(* CODESYS project cryo.library
   Placeholder: ESO LDC Cryo Library
   Title: ESO LDC Cryo Library
   Version: 0.0.0.10
   Company: ESO

Project tree, tasks and I/O mapping:
  libraries: ESO LDC Comm Common Library, 0.2.0.2 (ESO); ESO LDC Comm Serial Library, 0.2.0.2 (ESO); ESO LDC Comm Tcp Library, * (ESO); Tc2_SerialCom, * (Beckhoff Automation GmbH); Tc2_Standard, * (Beckhoff Automation GmbH); Tc2_System, * (Beckhoff Automation GmbH); Tc2_Utilities, * (Beckhoff Automation GmbH); Tc3_Module, * (Beckhoff Automation GmbH); VisuDialogs, * (System); VisuSymbols, 3.5.10.0 (System)
  config/
    CPA_Mapping_SPLC016.xml
    IRATEC_Mapping.xml
    MICADO_Mapping_Evacuation_Local.xml
    SIM_Mapping.xml
  00000000-0000-0000-0000-000000000000|config\CPA_Mapping_SPLC016.xml
  00000000-0000-0000-0000-000000000000|config\IRATEC_Mapping.xml
  00000000-0000-0000-0000-000000000000|config\MICADO_Mapping_Evacuation_Local.xml
  00000000-0000-0000-0000-000000000000|config\SIM_Mapping.xml
  DUTs/
    Enumerations/
      Actuators/
        data type E_CRYO_BIN_ACT_CMD
        data type E_CRYO_BIN_ACT_FEEDBACK
        data type E_CRYO_BIN_ACT_FEEDBACK_STATE
        data type E_CRYO_BIN_ACT_STATE
        data type E_CRYO_BIN_CTRL_ACTION
        data type E_CRYO_BIN_CTRL_STATE
        data type E_CRYO_CTRL_CMD
        data type E_CRYO_CTRL_STATE
        data type E_CRYO_GEN_CTRL_EVENT
      Coolers/
        data type E_CRYO_CPA_ALARM
        data type E_CRYO_CPA_CMDS
        data type E_CRYO_CPA_DIAG_IDX
        data type E_CRYO_CRYOTELGT_CMD
        data type E_CRYO_CRYOTELGT_STATE
      Misc/
        data type E_CRYO_ALARM_IDX
        data type E_CRYO_ALARM_LEVEL
        data type E_CRYO_THLD_MODE
        data type E_CRYO_VOTE
      Pumps/
        data type E_CRYO_PUMP_STATE
        data type E_ECODRY_VERSION
      Sensors/
        data type E_CRYO_SBG232_SENSOR_TYPE
        data type E_CRYO_SENSOR_TYPE_PRESS
        data type E_CRYO_SENSOR_TYPE_TEMP
        data type E_CRYO_SIM_SENS_CMD
      Subsystems/
        Evacuation/
          data type E_CRYO_EVAC_PRESSURES_50000
          data type E_CRYO_EVAC_STATE
          data type E_CRYO_EVAC_STATE_50000
          data type E_CRYO_EVAC_SYS_STATE
          data type E_CRYO_EVAC_VALVES_50000
    Structures/
      Actuators/
        data type T_CRYO_BIN_ACT_STATUS
        data type T_CRYO_BIN_CTRL_STATUS
        data type T_CRYO_GEN_CTRL_STATUS_BASE
      Coolers/
        data type T_CRYO_CPA_ACTIVE_LIMITS
        data type T_CRYO_CPA_CFG
        data type T_CRYO_CPA_CTRL
        data type T_CRYO_CPA_DIAG_CFG
        data type T_CRYO_CPA_INFO
        data type T_CRYO_CPA_STAT
        data type T_CRYO_CRYOTELGT_CFG
        data type T_CRYO_CRYOTELGT_CMD
        data type T_CRYO_CRYOTELGT_CTRL
        data type T_CRYO_CRYOTELGT_STAT
      Misc/
        data type T_CRYO_VOTE_LIST
      Pumps/
        data type T_CRYO_PUMP_ATM2303M_CFG
        data type T_CRYO_PUMP_ATM2303M_STAT
        data type T_CRYO_PUMP_BASE_CFG
        data type T_CRYO_PUMP_BASE_CTRL
        data type T_CRYO_PUMP_BASE_STAT
        data type T_CRYO_PUMP_CMD
        data type T_CRYO_PUMP_HIPACE30_CFG
        data type T_CRYO_PUMP_HIPACE30_STAT
        data type T_CRYO_PUMP_MODBUS_CFG
        data type T_CRYO_PUMP_MODBUS_CTRL
        data type T_CRYO_PUMP_MODBUS_STAT
        data type T_CRYO_PUMP_MVP030_CFG
        data type T_CRYO_PUMP_MVP030_STAT
        data type T_CRYO_PUMP_SERIAL_CFG
      Sensors/
        data type T_CRYO_IOLINK_SENSOR_STATUS
        data type T_CRYO_PRESSURE_STATUS
        data type T_CRYO_PRESSURE_VOTE_STATUS
        data type T_CRYO_PT100_OHM2C_REC
        data type T_CRYO_SBG232_STAT
        data type T_CRYO_SENSOR_STATUS
        data type T_CRYO_SENSOR_STATUS_PRESS
        data type T_CRYO_SENSOR_STATUS_TEMP
        data type T_CRYO_TEMPERATURE_STATUS
      Subsystems/
        Evacuation/
          data type T_CRYO_EVAC_CFG
          data type T_CRYO_EVAC_CFG_50000
          data type T_CRYO_EVAC_CTRL
          data type T_CRYO_EVAC_CTRL_50000
          data type T_CRYO_EVAC_STAT
          data type T_CRYO_EVAC_STAT_50000
          data type T_CRYO_EVAC_SYS_INPUT
          data type T_CRYO_EVACUATION_SYSTEM_STATUS
      System/
        data type T_CRYO_CFG
        data type T_CRYO_CTRL
        data type T_CRYO_LOG
        data type T_CRYO_STAT
  GVLs/
  POUs/
    Actuators/
      function block FB_CRYO_ACTUATOR_CMD [ST]: M_SetPermissionOff, M_SetPermissionOn, M_SetPermissions
      function block FB_CRYO_BIN_ACT [ST]: M_GetFeedback, M_SetCtrlOutput, M_SetStatus
      function block FB_CRYO_BIN_CTRL [ST]: M_Reset, M_SetStatus, M_User_SetAction, M_User_TryRecovery
      function block FB_CRYO_CCC_CTRL [ST]: M_User_SetAction
      function block FB_CRYO_CMD_OVERRIDE [ST]: M_SetAllPermitted, M_SetPermissionOff, M_SetPermissionOn, M_SetPermissions
      function block FB_CRYO_GEN_CTRL_BASE [ST]: M_ActionOffExecute, M_ActionOnExecute, M_ActivitySwitchingOff, M_ActivitySwitchingOn, M_CheckForEvents, M_Configure, M_ControlLoop, M_ExecuteActuators, M_IsError, M_ProcessEvents, M_ReadInputs, M_SetStatus
      function block FB_CRYO_HEATER_CTRL [ST]: M_User_SetAction
      function block FB_CRYO_LN2_CTRL [ST]: M_SetStatus, M_User_SetAction
      function block FB_CRYO_VALVE_CTRL [ST]: M_SetStatus, M_User_SetAction
    Comm/
      function block FB_MODBUS_COMM_CPA [ST]
    Coolers/
      function block FB_CRYO_CPA [ST]: ActivityInitializing, ActivityMonitoring, CheckForEvents, M_ByteSwapFLOAT, M_ByteSwapINT, M_CheckDiagnostics, M_CheckErrors, M_CheckService, M_CheckWarnings, M_ExtractReadings, M_GetModelNumber, M_GetOperatingState, M_SetAlarmText, M_UserConfigure
      function block FB_CRYO_CRYOTELGT [ST]: ActivityInitializing, ActivityInitializing_new, ActivityMonitoring, M_AddCtrlCommands, M_ClearCtrlCommands, M_Configure, M_ExecuteComm, M_FindReadCommand, M_GetCouplerState, M_ReadFromReply, M_StateMachine, M_UpdateStatus, ProcessEvents
      function block FB_RS_COMM_CRYOTELGT [ST]: M_ActionInitExecute, M_ComPortControl, M_Reset
      function block FB_SIM_RS_COMM_CRYOTELGT [ST]: M_ActivityDo, M_GetSimReply
    Pumps/
      function block FB_CRYO_PUMP_ATH2303M [ST]: M_Configure, M_GetSpeed, M_IsReady, M_IsRunning, M_ReadFromReply, M_UpdateStatus
      function block FB_CRYO_PUMP_BASE [ST]: ActivityInitializing, ActivityMonitoring, CheckForEvents, M_Configure, M_ExecuteComm, M_GetCouplerState, M_GetSpeed, M_IsReady, M_IsRunning, M_StateMachine, M_UpdateStatus, ProcessEvents
      function block FB_CRYO_PUMP_ECODRY [ST]: M_Configure, M_ExtractReadings_V01, M_ExtractReadings_V21_22, M_IsReady, M_IsRunning, M_ReadFromReply, M_UpdateStatus
      function block FB_CRYO_PUMP_HIPACE30 [ST]: M_Configure, M_GetSpeed, M_IsReady, M_IsRunning, M_ReadFromReply, M_UpdateStatus
      function block FB_CRYO_PUMP_MODBUS [ST]: ActivityInitializing, ActivityMonitoring, M_ByteSwapFLOAT, M_ByteSwapINT, M_ByteSwapUINT, M_ExecuteComm, M_GetCouplerState, M_ReadFromReply, M_SetCommand
      function block FB_CRYO_PUMP_MVP030 [ST]: M_Configure, M_GetSpeed, M_IsReady, M_IsRunning, M_ReadFromReply, M_UpdateStatus
      function block FB_CRYO_PUMP_SERIAL [ST]: ActivityInitializing, ActivityMonitoring, M_ExecuteComm, M_GetCouplerState, M_PVP_Checksum, M_ReadFromReply
    Sensors/
      function block FB_CRYO_PRESSURE [ST]: M_ReadSensors, M_SetStatus
      function block FB_CRYO_PRESSURE_VOTE [ST]: M_CheckWarnings, M_Configure, M_SetConnected, M_SetStatus, M_SetStatus_Average, M_SetStatus_FirstValid, M_SetStatus_Maximum, M_SetStatus_Minimum, M_SetStatus_XooY, M_SetWarning
      function block FB_CRYO_SBG232 [ST]: M_Configure, M_SetError, M_SetReading, M_UpdateStatus
      function block FB_CRYO_SENSOR_BASE [ST]: M_ReadSensor, M_SetStatus
      function block FB_CRYO_SENSOR_PRESSURE [ST]: M_SetStatus, M_SetStatus_CMR_361, M_SetStatus_PKR_250, M_SetStatus_PKR_360, M_SetStatus_WRG_D_NW25
      function block FB_CRYO_SENSOR_TEMPERATURE [ST]: M_GetRamp, M_PT100_Interpolate_Ohm2C, M_PT100_Ohm2C, M_SetStatus, M_SetStatus_PT100
      function block FB_CRYO_TEMPERATURE [ST]: M_GetTemperatureFromLakeshore, M_ReadSensors, M_SetStatus
    Simulation/
      function block FB_CRYO_SIM_CTRL [ST]
      function block FB_CRYO_SIM_PRESSURE [ST]: M_bit2mbar, M_mbar2bit, M_RampTo, M_SetValue, M_StartCurve, M_StartRamp, M_Stop
      function block FB_CRYO_SIM_SBG232 [ST]
      function block FB_CRYO_SIM_SINE [ST]
      function block FB_CRYO_SIM_TEMPERATURE [ST]: M_bit2degK, M_degK2bit, M_RampTo, M_SetValue, M_StartRamp, M_StartSine, M_Stop
      function block FB_SIM_MODBUS_COMM_CPA [ST]: M_GetSimReply
    Subsystems/
      Evacuation/
        function block FB_CRYO_EVAC_BASE [ST]: M_Activity_ClosingValve, M_Activity_DelayBeforeStoppingPumps, M_Activity_Evacuating, M_Activity_Off, M_Activity_OpeningValve, M_Activity_StartingRoughingPump, M_Activity_StartingTurboPump, M_Activity_StoppingRoughingPump, M_Activity_StoppingTurboPump, M_Activity_WaitingCryoVacuum, M_Activity_WaitingPrevacuum, M_Activity_WaitingTurboPump2Stop, M_Configure, M_ExecuteControllers, M_GotoOff, M_ReadSensors, M_SetError, M_SetLabels, M_StateMachine, M_UpdateStatus
        function block FB_CRYO_EVAC_BASE_50000 [ST]: M_ActionExecute, M_Activity_ClosingAllValves, M_Activity_ClosingValve, M_Activity_DelayBeforeStoppingPumps, M_Activity_Evacuating, M_Activity_Off, M_Activity_OpeningValve, M_Activity_StartingPVP, M_Activity_StartingTMP, M_Activity_StoppingPVP, M_Activity_StoppingTMP, M_Activity_Waiting2Pressures, M_Activity_WaitingPressure, M_Activity_WaitingTMP2Stop, M_Configure, M_ExecuteControllers, M_ReadSensors, M_SetError, M_SetLabels, M_SetNextState, M_StateMachine, M_UpdateStatus
        function block FB_CRYO_EVACUATION_SYSTEM [ST]: M_CheckErrors, M_PumpCtrl, M_SetStatus, M_SetValveCommand, M_StateMachine, M_TrgValveClosure, M_User_TryRecovery
      Examples/
        Evacuation/
          function block FB_CRYO_EVAC_ECODRY_ATH2303M [ST]: M_Configure, M_ExecuteControllers
          function block FB_CRYO_EVAC_MICADO [ST]: M_Configure, M_ExecuteControllers
          function block FB_CRYO_EVAC_PDS [ST]: M_Configure, M_ExecuteControllers
          function block FB_SIM_MICADO_PUMPS [ST]
          function block FB_SIM_MICADO_VALVES [ST]
        LN2_Precooling/
          function block FB_CRYO_LN2_PRECOOL [ST]: M_ActionOffExecute, M_ActionOnExecute, M_ActivitySwitchingOff, M_ActivitySwitchingOn, M_Configure, M_ControlLoop, M_ExecuteActuators, M_IsError, M_SetStatus
          function block FB_SIM_LN2_PRECOOL [ST]
    System/
      function block FB_CRYO_CTRL [ST]: M_CheckForCommands, M_CheckForSensorErrors, M_CheckLakeshoreCommand, M_CheckVacuum, M_Configure, M_ExecuteControllers, M_GetHighestTemperature, M_GetLowestTemperature, M_GetState, M_ReadSensors, M_SafetyCheck, M_SetStatus, M_StateMachine, M_SysLog
    Utilities/
      function block FB_CRYO_THLD_BASE [ST]: M_CheckAlarms, M_GetHysteresis, M_SetThresholds, M_UserSetActiveThresholds, M_UserSetLabel
    program MAIN [ST]
  VISUs/
    GUIs/
      visualisation GUI_ATH2303M_EVAC_LAB
      visualisation GUI_CMD_OVERRIDE
      visualisation GUI_CPA
      visualisation GUI_CRYO
      visualisation GUI_CRYOTELGT
      visualisation GUI_ECODRY_V01_EVAC_LAB
      visualisation GUI_EVAC_LAB
      visualisation GUI_EVAC_MICADO
      visualisation GUI_EVAC_PDS
      visualisation GUI_HIPACE_30_EVAC_PDS
      visualisation GUI_IRATEC
      visualisation GUI_MICADO_Valves
      visualisation GUI_MVP030_EVAC_PDS
      visualisation GUI_P2_OVERRIDE
      visualisation GUI_Pressures
      visualisation GUI_PVV1_CMD
      visualisation GUI_SBG232
      visualisation GUI_SBG232_SIM
      visualisation GUI_T2_OVERRIDE
    Templates/
      visualisation GUI_TEMPLATE_ACTUATOR_CMD
      visualisation GUI_TEMPLATE_ACTUATOR_ENG
      visualisation GUI_TEMPLATE_ATH2303M
      visualisation GUI_TEMPLATE_CMD_OVERRIDE
      visualisation GUI_TEMPLATE_CRYO_CPA
      visualisation GUI_TEMPLATE_CRYO_EVAC_BASE
      visualisation GUI_TEMPLATE_CRYOTELGT
      visualisation GUI_TEMPLATE_ECODRY_V01
      visualisation GUI_TEMPLATE_HIPACE_30
      visualisation GUI_TEMPLATE_MVP030
      visualisation GUI_TEMPLATE_PRESS_OVERRIDE
      visualisation GUI_TEMPLATE_SBG232
      visualisation GUI_TEMPLATE_SENSOR_SIM_OVERRIDE
      visualisation GUI_TEMPLATE_TEMP_OVERRIDE
  ClassDiagram
  ClassDiagram_All
  ClassDiagram_Sensors
  text list GlobalTextList
  image pool ImagePool
  00000000-0000-0000-0000-000000000000|\\winhome\home\dpopovic\My Pictures\Cryo GUI Background 2500-50000L.PNG
*)

// DUTs/Enumerations/Actuators/E_CRYO_BIN_ACT_CMD
{attribute 'qualified_only'}
{attribute 'strict'}
TYPE E_CRYO_BIN_ACT_CMD :
(
	NONE	:= 0,
	OFF 	:= 1,
	ON		:= 2
);
END_TYPE

// DUTs/Enumerations/Actuators/E_CRYO_BIN_ACT_FEEDBACK
{attribute 'qualified_only'}
{attribute 'strict'}
TYPE E_CRYO_BIN_ACT_FEEDBACK :
(
	ON_AND_OFF	:= 0,	// There are two separate signals: ON (i_bON) and OFF (i_bOFF)
	ON_ONLY 	:= 1	// Feedback exists only for ON signal
);
END_TYPE

// DUTs/Enumerations/Actuators/E_CRYO_BIN_ACT_FEEDBACK_STATE
{attribute 'qualified_only'}
{attribute 'strict'}
TYPE E_CRYO_BIN_ACT_FEEDBACK_STATE :
(
	OFF		:= 0,
	ON	 	:= 1,
	ERROR	:= 2
);
END_TYPE

// DUTs/Enumerations/Actuators/E_CRYO_BIN_ACT_STATE
{attribute 'qualified_only'}
{attribute 'strict'}
TYPE E_CRYO_BIN_ACT_STATE :
(
	NONE := 0,
	OFF,
	SWITCHING_ON,
	ON,
	SWITCHING_OFF,
	ERROR
);
END_TYPE

// DUTs/Enumerations/Actuators/E_CRYO_BIN_CTRL_ACTION
TYPE E_CRYO_BIN_CTRL_ACTION :
(
	NONE := 0,
	OFF,
	ON
);
END_TYPE

// DUTs/Enumerations/Actuators/E_CRYO_BIN_CTRL_STATE
{attribute 'qualified_only'}
{attribute 'strict'}
TYPE E_CRYO_BIN_CTRL_STATE :
(
	NONE := 0,
	OFF,					// Controller OFF, Actuator OFF
	ACTIVE_SWITCHING_ON,	// Activating Controller
	ACTIVE_OFF,				// Controller active, Actuator OFF
	ACTIVE_ON,				// Controller active, Actuator ON
	ACTIVE_SWITCHING_OFF,	// Switching Actuator OFF and going OFF with Controller
	ERROR					// Actuator failure
);
END_TYPE

// DUTs/Enumerations/Actuators/E_CRYO_CTRL_CMD
{attribute 'qualified_only'}
{attribute 'strict'}
TYPE E_CRYO_CTRL_CMD :
(
	NONE	:= 0,
	PRECOOL,
	COOL,
	WARM_UP,
	REPRESSURIZE
);
END_TYPE

// DUTs/Enumerations/Actuators/E_CRYO_CTRL_STATE
{attribute 'qualified_only'}
{attribute 'strict'}
TYPE E_CRYO_CTRL_STATE :
(
	NONE 			:= 0,
	WARM_PRESS,				// Warm & Pressurized
	WARM_VACUUM,			// Warm & Vacuum
	PRE_COOLING,			// Pre_cooling
	PRE_COOLED,				// Pre_cooled
	COOLING_DOWN,			// Cooling down
	COLD,					// Cold, i.e. fully operational
	WARMING_UP,				// Warming up
	REPRESSURIZING,			// Re-pressurizing			
	ERROR					// Controller failure
);
END_TYPE

// DUTs/Enumerations/Actuators/E_CRYO_GEN_CTRL_EVENT
{attribute 'qualified_only'}
{attribute 'strict'}
TYPE E_CRYO_GEN_CTRL_EVENT :
(
	NONE := 0,
	ENABLE,
	DISABLE,
	OFF,
	IS_OFF,
	ON,
	IS_ON,
	ERROR
);
END_TYPE

// DUTs/Enumerations/Coolers/E_CRYO_CPA_ALARM
{attribute 'qualified_only'}
{attribute 'strict'}
TYPE E_CRYO_CPA_ALARM :
(
	NONE := 0,
	LOW,
	HIGH
);
END_TYPE

// DUTs/Enumerations/Coolers/E_CRYO_CPA_CMDS
{attribute 'qualified_only'}
{attribute 'strict'}
TYPE E_CRYO_CPA_CMDS :
(
	NONE	:= 0,
	START	:= 21,
	STOP
);
END_TYPE

// DUTs/Enumerations/Coolers/E_CRYO_CPA_DIAG_IDX
{attribute 'qualified_only'}
{attribute 'strict'}
TYPE E_CRYO_CPA_DIAG_IDX :
(
	WATER_IN	:= 0,
	WATER_OUT,
	OIL_TEMP,
	HELIUM_TEMP,
	HELIUM_LOW_PRESS_OP,
	HELIUM_HIGH_PRESS_OP,
	HELIUM_DELTA_PRESS,
	HELIUM_STATIC_LOW_PRESS,
	HELIUM_STATIC_HIGH_PRESS
);
END_TYPE

// DUTs/Enumerations/Coolers/E_CRYO_CRYOTELGT_CMD
{attribute 'qualified_only'}
{attribute 'strict'}
TYPE E_CRYO_CRYOTELGT_CMD :
(
	NONE := 0,
	OFF,
	ON,
	SET_POWER
);
END_TYPE

// DUTs/Enumerations/Coolers/E_CRYO_CRYOTELGT_STATE
{attribute 'qualified_only'}
{attribute 'strict'}
TYPE E_CRYO_CRYOTELGT_STATE :
(
	OFF := 0,
	STARTING,
	ON,
	STOPPING,
	ERROR
);
END_TYPE

// DUTs/Enumerations/Misc/E_CRYO_ALARM_IDX
{attribute 'qualified_only'}
{attribute 'strict'}
TYPE E_CRYO_ALARM_IDX :
(
	ALARM_LOW 		:= 1,
	WARNING_LOW		:= 2,
	WARNING_HIGH	:= 3,
	ALARM_HIGH		:= 4
);
END_TYPE

// DUTs/Enumerations/Misc/E_CRYO_ALARM_LEVEL
{attribute 'qualified_only'}
{attribute 'strict'}
TYPE E_CRYO_ALARM_LEVEL :
(
	ALARM_LOW 		:= -2,
	WARNING_LOW		:= -1,
	NORMAL			:= 0,
	WARNING_HIGH	:= 1,
	ALARM_HIGH		:= 2
);
END_TYPE

// DUTs/Enumerations/Misc/E_CRYO_THLD_MODE
{attribute 'qualified_only'}
{attribute 'strict'}
TYPE E_CRYO_THLD_MODE :
(
	FIXED := 0,		// Thresholds as set with input parameters
	ACTIVE,			// Thresholds are calculated based on input parameter(s)
	LAST_ACTIVE		// Thresholds are kept at last ACTIVE levels 
);
END_TYPE

// DUTs/Enumerations/Misc/E_CRYO_VOTE
{attribute 'qualified_only'}
{attribute 'strict'}
TYPE E_CRYO_VOTE :
(
	V_AVE	:= 0,
	V_MIN,
	V_MAX,
	V_1oo2,
	V_2oo3,
	V_3oo5
);
END_TYPE

// DUTs/Enumerations/Pumps/E_CRYO_PUMP_STATE
{attribute 'qualified_only'}
{attribute 'strict'}
TYPE E_CRYO_PUMP_STATE :
(
	OFF := 0,
	STARTING,
	ON,
	STOPPING,
	ERROR
);
END_TYPE

// DUTs/Enumerations/Pumps/E_ECODRY_VERSION
{attribute 'qualified_only'}
{attribute 'strict'}
TYPE E_ECODRY_VERSION :
(
	V01 := 0,
	V21_22
);
END_TYPE

// DUTs/Enumerations/Sensors/E_CRYO_SBG232_SENSOR_TYPE
{attribute 'qualified_only'}
{attribute 'strict'}
TYPE E_CRYO_SBG232_SENSOR_TYPE :
(
	NONE := 0,
	FLOW,
	TEMP
);
END_TYPE

// DUTs/Enumerations/Sensors/E_CRYO_SENSOR_TYPE_PRESS
{attribute 'qualified_only'}
{attribute 'strict'}
TYPE E_CRYO_SENSOR_TYPE_PRESS :
(
	NONE 		:= 0,
	PKR_250		:= 1,	// Pfeiffer PKR250 & PKR251 have the same formula
	CMR_361		:= 2,	// Pfeiffer CMR361
	WRG_D_NW25	:= 3,	// Edwards WRG-D-NW25
	PKR_360		:= 4	// Pfeiffer PKR360
);
END_TYPE

// DUTs/Enumerations/Sensors/E_CRYO_SENSOR_TYPE_TEMP
{attribute 'qualified_only'}
{attribute 'strict'}
TYPE E_CRYO_SENSOR_TYPE_TEMP :
(
	NONE 	:= 0,
	PT100	:= 1
);
END_TYPE

// DUTs/Enumerations/Sensors/E_CRYO_SIM_SENS_CMD
{attribute 'qualified_only'}
{attribute 'strict'}
TYPE E_CRYO_SIM_SENS_CMD :
(
	NONE	:= 0,
	SET 	:= 1,	// Set value
	RAMP	:= 2,	// Ramp value
	SINE	:= 3	// Vary value as SINE signal
);
END_TYPE

// DUTs/Enumerations/Subsystems/Evacuation/E_CRYO_EVAC_PRESSURES_50000
{attribute 'qualified_only'}
{attribute 'strict'}
TYPE E_CRYO_EVAC_PRESSURES_50000 :
(
	NONE := 0,
	VAG1,		
	VAG2,		
	VAG3,		
	VAGF,		
	VAGG		
);
END_TYPE

// DUTs/Enumerations/Subsystems/Evacuation/E_CRYO_EVAC_STATE
{attribute 'qualified_only'}
{attribute 'strict'}
TYPE E_CRYO_EVAC_STATE :
(
	NONE := 0,				// Undefined state.
	OFF,					// Everything is OFF.
	START_R_PUMP,			// Starting Roughing Pump.
	WAIT_PREVAC,			// Waiting for the prevaccum pressure to be reached.
	OPEN_INSULATION_VALVE,	// Opening Insulation Valve.
	START_T_PUMP,			// Starting Turbo-Molecular Pump.
	WAIT_CRYO_VAC,			// Waiting for the cryo pressure to drop below threshold.
	EVACUATING,				// System is running. Evacuation in progress.
	CLOSE_INSULATION_VALVE,	// Closing Insulation Valve.
	DELAY_STOPPING,			// Delay after closing Insulation valve before stopping pumps.
	STOP_T_PUMP,			// Stopping Turbo-Molecular Pump.
	STOP_R_PUMP,			// Stopping Roughing Pump.
	WAIT_T_PUMP_STOP		// Waiting for the Turbo-Molecular Pump to stop.
);
END_TYPE

// DUTs/Enumerations/Subsystems/Evacuation/E_CRYO_EVAC_STATE_50000
{attribute 'qualified_only'}
{attribute 'strict'}
TYPE E_CRYO_EVAC_STATE_50000 :
(
	NONE := 0,				// Undefined state.
	OFF,					// Everything is OFF.
	START_PVP,				// Starting PreVacuum Pump (Roughing Pump).
	OPEN_GBV,				// Opening gas-ballast valve
	WAIT_VAG3,				// Waiting for VAG3 pressure < 0.1 mbar.
	OPEN_PVV1,				// Opening PVV1 Pre-vacuum Valve.
	WAIT_VAG_1_3,			// Waiting for VAG1 & VAG3 pressure < 0.1 mbar.
	OPEN_PVV2,				// Opening PVV2 Pre-vacuum Valve.
	WAIT_VAG_F_G_1,			// Waiting for VAGF & VAGG pressure < 0.9x0.1 mbar.
	CLOSE_PVV2,				// Closing PVV2 Pre-vacuum Valve.
	CLOSE_PVV1,				// Closing PVV1 Pre-vacuum Valve.
	START_TMP,				// Starting Turbo-Molecular Pump (TMP).
	OPEN_PVV3,				// Opening PVV3 Pre-vacuum Valve.
	WAIT_VAG_2_3,			// Waiting for VAG2 & VAG3 pressure < 0.1 mbar.
	OPEN_PVV4,				// Opening PVV4 Pre-vacuum Valve.
	WAIT_VAG_F_G_2,			// Waiting for VAGF & VAGG pressure < 0.0001 mbar.
	CLOSE_GBV,				// Closing gas-ballast valve
	EVACUATING,				// System is running. Evacuation in progress.
	CLOSE_ALL_VALVES,		// Closing All Valves.
	DELAY_STOPPING,			// Delay after closing valves before stopping pumps.
	STOP_TMP_1,				// Stopping Turbo-Molecular Pump (TMP) - case 1.
	STOP_TMP_2,				// Stopping Turbo-Molecular Pump (TMP) - case 2.
	STOP_PVP,				// Stopping PreVacuum Pump (Roughing Pump).
	WAIT_TMP_STANDSTILL		// Waiting for the Turbo-Molecular Pump to standstill.
);
END_TYPE

// DUTs/Enumerations/Subsystems/Evacuation/E_CRYO_EVAC_SYS_STATE
{attribute 'qualified_only'}
{attribute 'strict'}
TYPE E_CRYO_EVAC_SYS_STATE :
(
	NONE := 0,
	OFF,					// Controller OFF, Valve closed
//	ACTIVE_STARTING_PUMPS,	// Controller ON,  Starting pumps
//	ACTIVE_PUMPS_RUNNING,	// Controller ON,  Pumps running
	ACTIVE_OPENING,			// Controller ON,  Valve opening
	ACTIVE_OPEN,			// Controller ON,  Valve open
	ACTIVE_CLOSING,			// Controller ON,  Valve closing
	ACTIVE_CLOSED,			// Controller ON,  Valve closed
//	ACTIVE_STOPPING_PUMPS,	// Controller ON,  Stopping pumps
	EMERGENCY,				// Controller ON,  Closing valve for safety reason
	ERROR					// Error in the system
);
END_TYPE

// DUTs/Enumerations/Subsystems/Evacuation/E_CRYO_EVAC_VALVES_50000
{attribute 'qualified_only'}
{attribute 'strict'}
TYPE E_CRYO_EVAC_VALVES_50000 :
(
	NONE := 0,
	PVV1,		
	PVV2,		
	PVV3,		
	PVV4,		
	GBV		
);
END_TYPE

// DUTs/Structures/Actuators/T_CRYO_BIN_ACT_STATUS
TYPE T_CRYO_BIN_ACT_STATUS :
STRUCT
	bDone:		BOOL;			// Flag if switch is OK
	bBusy:		BOOL;			// Flag if switch is BUSY
	bError:		BOOL;			// Flag if switch is OK
	bON:		BOOL;			// Flag if switch state is ON
	bOFF:		BOOL;			// Flag if switch state is OFF

	nLastCommand:	E_CRYO_BIN_ACT_CMD		:= E_CRYO_BIN_ACT_CMD.NONE;	// Command
	nState:			E_CRYO_BIN_ACT_STATE	:= E_CRYO_BIN_ACT_STATE.NONE;
	
	sState:		STRING(64);			// State as text
END_STRUCT
END_TYPE

// DUTs/Structures/Actuators/T_CRYO_BIN_CTRL_STATUS
TYPE T_CRYO_BIN_CTRL_STATUS :
STRUCT
	bDone:		BOOL;			// Flag if controller is OK
	bBusy:		BOOL;			// Flag if controller is BUSY
	bError:		BOOL;			// Flag if controller is OK
	bActive:	BOOL;			// Flag if controller is ACTIVE
	bActON:		BOOL;			// Flag if actuator is ON
	bActOFF:	BOOL;			// Flag if actuator is OFF

	// Generic controller OK flag.
	// Used for problems other than from the actuator.
	// This flag is used for problems coming from controllers
	// that extend the functionality of FB_CRYO_BIN_CTRL.
	bCtrlOK:	BOOL := TRUE;		

	nCycleCounter:	UDINT := 0;
	nState:			E_CRYO_BIN_CTRL_STATE	:= E_CRYO_BIN_CTRL_STATE.NONE;

	sState:		STRING(64);		// State as text
END_STRUCT
END_TYPE

// DUTs/Structures/Actuators/T_CRYO_GEN_CTRL_STATUS_BASE
TYPE T_CRYO_GEN_CTRL_STATUS_BASE :
STRUCT
	bDone:			BOOL;			// Flag if controller is OK
	bBusy:			BOOL;			// Flag if controller is BUSY
	bError:			BOOL;			// Flag if controller is in ERROR state
	bActive:		BOOL;			// Flag if controller is ACTIVE

	nCycleCounter:	UDINT := 0;
	nState:			E_CRYO_BIN_CTRL_STATE	:= E_CRYO_BIN_CTRL_STATE.NONE;

	sState:			STRING(64);		// State as text
	sError:			STRING(64);		// Error as text
END_STRUCT
END_TYPE

// DUTs/Structures/Coolers/T_CRYO_CPA_ACTIVE_LIMITS
TYPE T_CRYO_CPA_ACTIVE_LIMITS :
STRUCT
	rErrorLow:		REAL;	// Error for Low  range
	rAlarmLow:		REAL;	// Alarm for Low  range MAX(CRYOMECH,ESO)
	rAlarmHigh:		REAL;	// Alarm for High range MIN(CRYOMECH,ESO)
	rErrorHigh:		REAL;	// Error for High range
END_STRUCT
END_TYPE

// DUTs/Structures/Coolers/T_CRYO_CPA_CFG
TYPE T_CRYO_CPA_CFG EXTENDS T_RS_BASE_CFG:
STRUCT
	// Register Addresses
	nAddrCommon:		INT	:= 16#0001;	// 16#0001

	// Number of bytes to read
	// These are ONLY data bytes. Total bytes to read is higher (+5) 
	nWordsCommon:		INT	:= 32;	// 64w=128 bytes
	
	nSlaveID:			BYTE := 1;	// Slave ID
	bDevUsed:			BOOL := TRUE;	

	nPosOffset:	INT	:= 0;	// byte position in the buffer - for testing
	
	// Thresholds for 'service due' warnings.
	// Warning 'Service due in xxx hours' will appear if less than the threshold is left.
	lrServiceDue_Compressor:	LREAL	:= 1000.0; // hours
	lrServiceDue_PulseTube:		LREAL	:= 2000.0; // hours
	
	
//
// Alarms and warnings
//
	
(*
7.7.7 Error and warning set points
==================================
"High pressure too High!" YES 400 PSIG (27.6bar) 375 PSIG (25.9 bar)
"High pressure too Low!" YES 150 PSIG (10.3bar) 170 PSIG (11.7 bar)
“Low Pressure Too Low!” YES 40 PSIG (2.8 bar) 50 PSIG (3.4 bar)
“Low Pressure Too High!" YES 250 PSIG (17.2 bar) 240 PSIG (16.5 bar)
"Delta Pressure Too High!" YES 400 PSIG (27.6bar) 275 PSIG (19 bar)
"Delta Pressure Too Low!" YES 50 PSIG (3.4 bar) 75 PSIG (5.2 bar)
"Static Pressure Too High!" YES 300 PSIG (20.7 bar) 280 PSIG (19.3 bar)
"Static Pressure Too Low!" YES 100 PSIG (6.9 bar) 170 PSIG (11.7 bar)
"Water In Temp Too High" YES 110°F (43°C) 80°F (27°C)
"Water In Temp Too Low" YES 40°F (4°C) 50°F (10°C)
“Water Out Temp Too High!” YES 125°F (52°C) 110°F (43°C)
"Water Out Temp Too Low" YES 40°F (4°C) 50°F (10°C)
“Helium Temp Too High!” YES 190°F (88°C) 120°F (49°C)
“Helium Temp Too Low!" YES 40°F (4°C) 50°F (10°C)
“Oil Temp Too High!” YES 125°F (52°C) 110°F (43°C)
“Oil Temp Too Low!" YES 40°F (4°C) 50°F (10°C)
“Compressor Motor Current Too Low!” YES < 5A ≥ 5 A


Warning Description Trip / Clear
================================
"High Pressure Running High!" 375 PSIG (25.9bar)
"High Pressure Running Low!" 170 PSIG (11.7bar)
“Low Pressure Running Low!” 50 PSIG (3.4 bar)
“Low Pressure Running High!" 240 PSIG (16.5 bar)
"Delta Pressure Running High!" 275 PSIG (19.0bar)
"Delta Pressure Running Low!" 75 PSIG (5.2 bar)
"Static Pressure Running High!" 280 PSIG (19.3 bar)
"Static Pressure Running Low!" 170 PSIG (11.7 bar)
"Water In Temp Running High" 85°F (29°C)
"Water In Temp Running Low" 45°F (7°C)
“Water Out Temp Running High!” 110°F (43°C)
"Water Out Temp Running Low" 45°F (7°C)
“Helium Temp Running High!” 170°F (77°C)
“Helium Temp Running Low!" 45°F (7°C)
“Oil Temp Running High!” 110°F (43°C)
“Oil Temp Running Low!" 45°F (7°C)

*)
	//
	// Diagnostics configuration.
	// Low and high limits for alarms and errors.
	//
	aDiag:	ARRAY [0..8] OF T_CRYO_CPA_DIAG_CFG := [ 
		(sLabel:='Water IN',	sUnits:='ºC',	nBitLow:=1, nBitHigh:=0,
			rErrorLow:=4.0, 		rAlarmLow_CPA:=7.0,	rAlarmLow_ESO:=7.0,	
			rAlarmHigh_ESO:=27.0,	rAlarmHigh_CPA:=29.0,	rErrorHigh:=43.0),
		(sLabel:='Water OUT',	sUnits:='ºC', 	nBitLow:=3, nBitHigh:=2,
			rErrorLow:=4.0, 		rAlarmLow_CPA:=7.0, 	rAlarmLow_ESO:=7.0, 
			rAlarmHigh_ESO:=50.0, 	rAlarmHigh_CPA:=43.0, 	rErrorHigh:=52.0),
		(sLabel:='Oil temperature', sUnits:='ºC',  	nBitLow:=5, nBitHigh:=4,
			rErrorLow:=4.0, 		rAlarmLow_CPA:=7.0, 	rAlarmLow_ESO:=7.0, 
			rAlarmHigh_ESO:=50.0, 	rAlarmHigh_CPA:=43.0, 	rErrorHigh:=52.0),
		(sLabel:='Helium temperature', 				sUnits:='ºC',  	nBitLow:=7, nBitHigh:=6,
			rErrorLow:=4.0, 		rAlarmLow_CPA:=7.0, 	rAlarmLow_ESO:=7.0, 
			rAlarmHigh_ESO:=80.0, 	rAlarmHigh_CPA:=77.0, 	rErrorHigh:=88.0),
		(sLabel:='Operational Helium low pressure',	sUnits:='bar',  	nBitLow:=9, nBitHigh:=8,
			rErrorLow:=2.8, 		rAlarmLow_CPA:=3.4, 	rAlarmLow_ESO:=4.0, 
			rAlarmHigh_ESO:=13.0, 	rAlarmHigh_CPA:=16.5, 	rErrorHigh:=17.2),
		(sLabel:='Operational Helium high pressure',	sUnits:='bar',  	nBitLow:=11, nBitHigh:=10,
			rErrorLow:=10.3, 		rAlarmLow_CPA:=11.7, 	rAlarmLow_ESO:=17.0, 
			rAlarmHigh_ESO:=25.0, 	rAlarmHigh_CPA:=25.9, 	rErrorHigh:=27.6),
		(sLabel:='Delta operational Helium pressure',	sUnits:='bar',  	nBitLow:=13, nBitHigh:=12,
			rErrorLow:=3.4, 		rAlarmLow_CPA:=5.2, 	rAlarmLow_ESO:=6.0, 
			rAlarmHigh_ESO:=18.0, 	rAlarmHigh_CPA:=19.0, 	rErrorHigh:=27.6),
		(sLabel:='Static Helium low pressure',			sUnits:='bar',  	nBitLow:=18, nBitHigh:=17,
			rErrorLow:=6.9, 		rAlarmLow_CPA:=11.7, 	rAlarmLow_ESO:=12.0, 
			rAlarmHigh_ESO:=19.0, 	rAlarmHigh_CPA:=19.3, 	rErrorHigh:=20.7),
		(sLabel:='Static Helium high pressure',		sUnits:='bar',  	nBitLow:=18, nBitHigh:=17,
			rErrorLow:=6.9, 		rAlarmLow_CPA:=11.7, 	rAlarmLow_ESO:=12.0, 
			rAlarmHigh_ESO:=19.0, 	rAlarmHigh_CPA:=19.3, 	rErrorHigh:=20.7)];
	
	// Dynamic pressure limits.
	// Limits depend on compressor state 
	// ON 	- Operational pressure
	// OFF - Static pressure
//	stActPressLimit_Low:	T_CRYO_CPA_ACTIVE_LIMITS;
//	stActPressLimit_High:	T_CRYO_CPA_ACTIVE_LIMITS;
	// Array of limits. Dynamically set
	aLimits:	ARRAY [0..6] OF T_CRYO_CPA_ACTIVE_LIMITS;	
	aLimits_OP:	ARRAY [0..6] OF T_CRYO_CPA_ACTIVE_LIMITS;	
	aLimits_ST:	ARRAY [0..6] OF T_CRYO_CPA_ACTIVE_LIMITS;	

	

END_STRUCT
END_TYPE

// DUTs/Structures/Coolers/T_CRYO_CPA_CTRL
TYPE T_CRYO_CPA_CTRL EXTENDS T_RS_BASE_CTRL:
STRUCT
	nDevCommand:	E_CRYO_CPA_CMDS := E_CRYO_CPA_CMDS.NONE;	// CPA specific commands
	bCtrlPulseActive:	BOOL	:= FALSE;	// Switching compressor on/off active

	nSlaveID:	BYTE 	:= 1;						// Modbus Slave ID, 1..247
	nCmdType:	DINT	:= E_MODBUS_CMD_TYPE.READ;	// Command type; 0-Read, 1-Write
	nRegister:	DINT;								// Command register
	nWords:		DINT	:= 1;						// Number of words
	nValue:		DINT;								// Parameter value
	
	
END_STRUCT
END_TYPE

// DUTs/Structures/Coolers/T_CRYO_CPA_DIAG_CFG
TYPE T_CRYO_CPA_DIAG_CFG :
STRUCT
	sLabel:				STRING(56)	:= '';	// Label for Inputs, e.g. 'Water IN'
	sUnits:				STRING(8)	:= '';	// User units
	nBitLow:			INT;	// Bit position in warnings/errors for Low
	nBitHigh:			INT;	// Bit position in warnings/errors for High
	rErrorLow:			REAL;	// Error for Low  range
	rAlarmLow_CPA:		REAL;	// Alarm for Low  range as defined by CRYOMECH
	rAlarmLow_ESO:		REAL;	// Alarm for Low  range as defined by ESO
	rAlarmHigh_ESO:		REAL;	// Alarm for High range as defined by ESO
	rAlarmHigh_CPA:		REAL;	// Alarm for High range as defined by CRYOMECH
	rErrorHigh:			REAL;	// Error for High range
END_STRUCT
END_TYPE

// DUTs/Structures/Coolers/T_CRYO_CPA_INFO
TYPE T_CRYO_CPA_INFO :
STRUCT
(*
	Driver Information

	Change LOG:
*)
	sDate:			STRING(16)	:= '2020-07-14';
	sDescription:	STRING(32) 	:= 'CPA controller';
	sName:			STRING(16)	:= 'FB_CRYO_CPA';
	sPlatform:		STRING(16)	:= 'CoDeSys';
	sSynopsis:		STRING(48)	:= 'EtherCAT PLC CPA controller';
	nVersionMajor:	DINT		:= 1;
	nVersionMinor:	DINT		:= 0;

END_STRUCT
END_TYPE

// DUTs/Structures/Coolers/T_CRYO_CPA_STAT
TYPE T_CRYO_CPA_STAT EXTENDS T_RS_BASE_STAT:
STRUCT
	bSystemOn:				BOOL := FALSE;

	nRetries:				INT := 0;	// Total number of retries in case of communication problems
	
	nInputBuffer: 			ARRAY [0..300] OF BYTE;	// Binary data read from JUMO
	
	// Parameters read from the compressor
	nOperatingState:		INT	:= 0;
	nCompressorRunning:		INT	:= 0;
	lrWarningState:			LREAL	:= 0.0;
	lrAlarmState:			LREAL	:= 0.0;
	lrCoolantInTemp:		LREAL	:= 0.0;
	lrCoolantOutTemp:		LREAL	:= 0.0;
	lrOilTemp:				LREAL	:= 0.0;
	lrHeliumTemp:			LREAL	:= 0.0;
	lrLowPressure:			LREAL	:= 0.0;
	lrLowPressureAverage:	LREAL	:= 0.0;
	lrHighPressure:			LREAL	:= 0.0;
	lrHighPressureAverage:	LREAL	:= 0.0;
	lrDeltaPressureAverage:	LREAL	:= 0.0;
	lrMotorCurrent:			LREAL	:= 0.0;
	lrHoursOfOperation:		LREAL	:= 0.0;
	nPressureScale:			INT		:= 0;
	nTempScale:				INT		:= 0;
	nPanelSerialNumber:		UINT	:= 0;
	nModelMajorMinor:		INT		:= 0;

	// Calculated values
	sOperatingState:		STRING(32);
	sModelNumber:			STRING	:= 'CRYOMECH CPAxxxx';

	sServiceDue_Compressor:	STRING	:= ''; 		// Warning string for compressor service
	sServiceDue_PulseTube:	STRING	:= ''; 		// Warning string for pulse tube service
	

	bServiceDue_Compressor:	BOOL	:= FALSE;	// Warning for compressor service
	bServiceDue_PulseTube:	BOOL	:= FALSE;	// Warning for pulse tube service
	
	wColour_Compressor:		DWORD;	// Warning colour for compressor service
	wColour_PulseTube:		DWORD;	// Warning colour for pulse tube service

	
	
(*	
Input Register 30005: (Errors)
0: No Errors
-1: CoolantInHigh
-2: CoolantInLow
-4: CoolantOutHigh
-8: CoolantOutLow
-16: OilHigh
-32: OilLow
-64: HeliumHigh
-128: HeliumLow
-256: LowPressureHigh
-512: LowPressureLow
-1024: HighPressureHigh
-2048: HighPressureLow
-4096: DeltaPressureHigh
-8192: DeltaPressureLow
-16384: MotorCurrentLow
-32768: ThreePhaseError
-65536: PowerSupplyError
-131072: StaticPressureHigh
-262144: StaticPressureLow
*)
	
	
	// Readings in array
	aReadings:	ARRAY [0..6] OF LREAL;	// For index, see E_CRYO_CPA_DIAG_IDX
	
	// Alarms in array
	arrAlarms:		ARRAY [0..8] OF INT;
	// Errors in array
	arrErrors:		ARRAY [0..8] OF INT;
	
	// Alarm text, e.g. 
	// ‘Alarm: high pressure running high, compressor will shut off at 27.6 bar’
	sAlarm:		STRING(128)	:= '';	
	// Error text, e.g. 
	// ‘Error: high pressure running high, compressor shut off at 27.6 bar’
	sError:		STRING(128)	:= '';	
	sStatusOK:	STRING(128)	:= 'Running Normally';	
	
	nStatusCode:	INT	:= 0;	// 0-OK, 1-Alarm, 2-Error

	
END_STRUCT
END_TYPE

// DUTs/Structures/Coolers/T_CRYO_CRYOTELGT_CFG
TYPE T_CRYO_CRYOTELGT_CFG EXTENDS T_RS_BASE_CFG:
STRUCT

	tDelay_Read:		TIME 	:= T#150MS;	// Delay between sending each cmdList_Read[] command.
	nTimeoutState:		UDINT	:= 60000;	// 60 sec default timeout for starting and stopping cooler

	cmdList_Init:	ARRAY [1..8] OF T_CRYO_CRYOTELGT_CMD := [
		(cmd := 'VERSION', 				nReplies := 2),	// Current controller code version
		(cmd := 'MODE', 				nReplies := 2),	// MODE Cryocooler type, e.g. GT
		(cmd := 'SENSOR', 				nReplies := 2),	// Configured temp. sensor type, e.g. 'PT-100'
		(cmd := 'PWOUT=240', 			nReplies := 2),	// Set commanded power to 240 W
		(cmd := '', 					nReplies := 0),
		(cmd := '', 					nReplies := 0),
		(cmd := '', 					nReplies := 0),
		(cmd := '', 					nReplies := 0)];
	
	cmdList_Read:	ARRAY [1..16] OF T_CRYO_CRYOTELGT_CMD := [
		(cmd := 'ERROR', 				nReplies := 2),	// Controller error flags
		(cmd := 'COOLER', 				nReplies := 2),	// Cooler control mode, e.g. POWER or OFF
		(cmd := 'P', 					nReplies := 2),	// Measured cryocooler power
		(cmd := 'PWOUT', 				nReplies := 2),	// User commanded power
		(cmd := 'TC', 					nReplies := 2),	// Temperature sensor reading [K]
		(cmd := 'TEMP RJ', 				nReplies := 2),	// Reject temperature in [C]
		(cmd := '', 					nReplies := 0),
		(cmd := '', 					nReplies := 0),
		(cmd := '', 					nReplies := 0),
		(cmd := '', 					nReplies := 0),
		(cmd := '', 					nReplies := 0),
		(cmd := '', 					nReplies := 0),
		(cmd := '', 					nReplies := 0),
		(cmd := '', 					nReplies := 0),
		(cmd := '', 					nReplies := 0),
		(cmd := '', 					nReplies := 0)];
	

END_STRUCT
END_TYPE

// DUTs/Structures/Coolers/T_CRYO_CRYOTELGT_CMD
TYPE T_CRYO_CRYOTELGT_CMD :
STRUCT
	cmd:		STRING	:= '';	// Command to send
	nReplies:	INT	:= 1;	// # of Replies
END_STRUCT
END_TYPE

// DUTs/Structures/Coolers/T_CRYO_CRYOTELGT_CTRL
TYPE T_CRYO_CRYOTELGT_CTRL EXTENDS T_RS_BASE_CTRL:
STRUCT
	nDevCmd:	E_CRYO_CRYOTELGT_CMD := E_CRYO_CRYOTELGT_CMD.NONE;
	bStart:		BOOL;			// Control to Start/Stop the cooler.
	bPower:		BOOL;			// Update cooler power output.
	lrPower:	LREAL:= 240.0;	// Output power to set [W]
END_STRUCT
END_TYPE

// DUTs/Structures/Coolers/T_CRYO_CRYOTELGT_STAT
TYPE T_CRYO_CRYOTELGT_STAT EXTENDS T_RS_BASE_STAT :
STRUCT
	
	nRetries:			UDINT := 0;			// Total number of retries in case of communication problems
	nDevState:			E_CRYO_CRYOTELGT_STATE := E_CRYO_CRYOTELGT_STATE.OFF;
	sDevState:			STRING := 'OFF';

	sReply:				STRING(255); 		(* Last Reply to predefined commands*)

	// Status attributes that are read from the controller via RS-232
	sVersion:			STRING;
	sMode:				STRING;
	sSensor:			STRING;
	sCtrlError:			STRING;
	sCtrlMode:			STRING;
	
	lrPowerMeasured:	LREAL;
	lrPowerCommanded:	LREAL;
	lrTempColdHead:		LREAL;
	lrTempReject:		LREAL;
	lrTempTarget:		LREAL;
	
	bPowerCmdActive:	BOOL;
	
END_STRUCT
END_TYPE

// DUTs/Structures/Misc/T_CRYO_VOTE_LIST
// This structure is used to keep indexes of minimal reading differences
TYPE T_CRYO_VOTE_LIST :
STRUCT
	nIndex1:	INT;
	nIndex2:	INT;
	lrValue:	LREAL;	
END_STRUCT
END_TYPE

// DUTs/Structures/Pumps/T_CRYO_PUMP_ATM2303M_CFG
TYPE T_CRYO_PUMP_ATM2303M_CFG EXTENDS T_CRYO_PUMP_SERIAL_CFG:
STRUCT
// TODO: Add specific configuration here

	// Definition of commands
	C_CMD_NONE:		STRING(16) := '';
	C_CMD_IDN:		STRING(16) := '#000IDN';
	C_CMD_RDI:		STRING(16) := '#000RDI';
	C_CMD_VER:		STRING(16) := '#000VER';
	C_CMD_DEF:		STRING(16) := '#000DEF';
	C_CMD_SEL:		STRING(16) := '#000SEL10';
	C_CMD_TIM:		STRING(16) := '#000TIM';
	C_CMD_STA:		STRING(16) := '#000STA';
	C_CMD_LEV:		STRING(16) := '#000LEV10';

END_STRUCT
END_TYPE

// DUTs/Structures/Pumps/T_CRYO_PUMP_ATM2303M_STAT
TYPE T_CRYO_PUMP_ATM2303M_STAT EXTENDS T_CRYO_PUMP_BASE_STAT :
STRUCT

	// Digital status input signals
	bSpeed100:			BOOL;	// pump speed > 100 rpm
	
	
	// STA command
	// All attributes are defined in T_CRYO_PUMP_BASE_STAT
	
	// LEV10 command
	nNominalSpeed:				DINT;	// [rpm]
	nStandbySpeed:				DINT;	// [rpm]
	nSetPoint_AtSpeed:			DINT;	// ‘At speed’ relay set point (3 to 50%)
	nSetPoint_Temp:				DINT;	// temperature set point (30 to 65°C)
	nSetPoint_BearingWarn:		DINT;	// landing bearing warning set point (0 to 99%)
	nSetPoint_BearingCounter:	DINT;	// landing bearing counter (0 to 100%)
	
	// SEL command
	
	// VER Command (4 version strings)
	sVer1:	STRING;
	sVer2:	STRING;
	sVer3:	STRING;
	sVer4:	STRING;

	sIDN:	STRING;
	sRDI:	STRING;
	
	
END_STRUCT
END_TYPE

// DUTs/Structures/Pumps/T_CRYO_PUMP_BASE_CFG
TYPE T_CRYO_PUMP_BASE_CFG EXTENDS T_RS_BASE_CFG:
STRUCT

	nModel:				DINT := 0;			// Model 0 indicates the base FB.
	nTimeoutState:		UDINT	:= 600000;	// 600 sec default timeout for starting and stopping pump
	

END_STRUCT
END_TYPE

// DUTs/Structures/Pumps/T_CRYO_PUMP_BASE_CTRL
TYPE T_CRYO_PUMP_BASE_CTRL EXTENDS T_RS_BASE_CTRL:
STRUCT
	bStart:		BOOL;	// Control to Start/Stop the pump.
END_STRUCT
END_TYPE

// DUTs/Structures/Pumps/T_CRYO_PUMP_BASE_STAT
TYPE T_CRYO_PUMP_BASE_STAT EXTENDS T_RS_BASE_STAT :
STRUCT
	
	nRetries:			UDINT := 0;			// Total number of retries in case of communication problems
	nPumpState:			E_CRYO_PUMP_STATE := E_CRYO_PUMP_STATE.OFF;
	sPumpState:			STRING := 'OFF';

	sReply:				STRING(255); 		(* Last Reply to predefined commands*)

	// Digital status input signals
	bReady:				BOOL;	// If TRUE, pump is operational
	bMoving:			BOOL;	// If TRUE, pump is rotating, i.e. speed > 0.
	bWarning:			BOOL;	// presence of a warning
	bAlarm:				BOOL;	// presence of an alarm
	
	// Values obtained via serial communication
	nCtrlMode:			DINT;	// e.g. 0-Hand held, 1-Remote, 2-Serial, etc
	sCtrlMode:			STRING;	// e.g. 'Hand held', 'Remote', 'Serial', etc

	bON:				BOOL;	// Flag if Motor Pump is ON
	nElecPower:			DINT;	// Electronic drive power [W]
	nElecHours:			DINT;	// Electronic drive unit operating hours
	nElecTemp:			DINT;	// Drive Electronics Temperature [degC]
	nMotorCurr:			DINT;	// Pump Motor Current [mA]
	nMotorVolt:			DINT;	// Pump Motor Voltage [V]
	nPumpHours:			DINT;	// Pump operating hours
	nPumpSpeed:			DINT;	// Pump Motor Speed [rpm]
	nPumpTemp:			DINT;	// Pump Temperature[degC]
	
	
	
END_STRUCT
END_TYPE

// DUTs/Structures/Pumps/T_CRYO_PUMP_CMD
TYPE T_CRYO_PUMP_CMD :
STRUCT
	cmd:	STRING	:= '';	// Command to send
	length:	DINT	:= 1;	// Reply length
END_STRUCT
END_TYPE

// DUTs/Structures/Pumps/T_CRYO_PUMP_HIPACE30_CFG
TYPE T_CRYO_PUMP_HIPACE30_CFG EXTENDS T_CRYO_PUMP_SERIAL_CFG:
STRUCT
// HIPACE30 specific command configuration.
// Pfeiffer Vacuum protocol for RS-485 interface.
// Assumed RS-485 device ID=1 (001) !!!

	// Definition of commands
	C_CMD_NONE:				STRING(16) := '';
	C_CMD_sCtrlViaInt:		STRING(16) := '0011006003001';	// Control via DIO
	C_CMD_sFwVersion:		STRING(16) := '0010031202=?';
	C_CMD_sHwVersion:		STRING(16) := '0010035402=?';
	C_CMD_nNominalSpeed:	STRING(16) := '0010039902=?';
	
	C_CMD_bON:				STRING(16) := '0010002302=?';
	C_CMD_nCtrlMode:		STRING(16) := '0010006002=?';
	C_CMD_sErrorCode:		STRING(16) := '0010030302=?';
	C_CMD_bTargetSpeed:		STRING(16) := '0010030602=?';
	C_CMD_nMotorCurr:		STRING(16) := '0010031002=?';
	C_CMD_nPumpHours:		STRING(16) := '0010031102=?';
	C_CMD_nMotorVolt:		STRING(16) := '0010031302=?';
	C_CMD_nElecHours:		STRING(16) := '0010031402=?';
	C_CMD_nElecTemp:		STRING(16) := '0010032602=?';
	C_CMD_nPumpTemp:		STRING(16) := '0010034602=?';
	C_CMD_nPumpSpeed:		STRING(16) := '0010039802=?';
	

END_STRUCT
END_TYPE

// DUTs/Structures/Pumps/T_CRYO_PUMP_HIPACE30_STAT
TYPE T_CRYO_PUMP_HIPACE30_STAT EXTENDS T_CRYO_PUMP_BASE_STAT :
STRUCT

(*
Type:
0 - old bool: 0=FALSE, NOT 0 = TRUE.
1 - UDINT
2 - REAL * 100 (with leading zeros), e.g. 001571 corresponds with 15.71
4 - STRING (6)
7 - UINT (000 to 999)

INIT commands
023 MotorPump Motor pump 0 = off 1 = on 0 RW 0 1 1
060 CtrlViaInt Control via interface 7 RW 1 255 1
	1 = remote 
	2 = RS-485 
	4 = PV.can
	8 = Fieldbus
	16 = E74
	255 = unlock interface selection

312 Fw version Firmware version electronic drive unit 4 R
354 HW Version Hardware version electronic drive unit 4 R

STATUS commands
303 Error code Error code 4 R
306 SetSpdAtt Target speed reached 0 = no 1 = yes 0 R 0 1
310 DrvCurrent Drive current 2 R A 0 9999.99
311 OpHrsPump Operating hours pump 1 R h 0 65535
313 DrvVoltage Drive voltage 2 R V 0 9999.99
314 OpHrsElec Operating hours electronic drive unit 1 R h 0 65535
316 *** DrvPower Drive power 1 R W 0 999999
319 *** PumpCycles Pump cycles 1 R 0 65535
326 TempElec Temperature electronics 1 R °C 0 999999
346 ^^^ TempMotor Temperature motor 1 R °C 0 999999
397 *** SetRotSpd Set rotation speed (rpm) 1 R rpm 0 999999
398 ActualSpd Actual rotation speed (rpm) 1 R rpm 0 999999
399 NominalSpd Nominal rotation speed (rpm) 1 R rpm 0 999999

*)

// INIT commands
	sFwVersion:		STRING(8);
	sHwVersion:		STRING(8);

// STATUS commands
	sFailureCode:	STRING(8) := 'OK';
	bTargetSpeed:	BOOL;		// Target Speed Reached
	nNominalSpeed:	DINT;		// [rpm] Nominal Pump Speed
	lrMotorVolt:	LREAL;		// Pump Motor Voltage [V]
	
	bFailure:		BOOL := FALSE;	// Err of Wrn (see cmd 303)
END_STRUCT
END_TYPE

// DUTs/Structures/Pumps/T_CRYO_PUMP_MODBUS_CFG
TYPE T_CRYO_PUMP_MODBUS_CFG EXTENDS T_CRYO_PUMP_BASE_CFG:
STRUCT
	nSlaveID:	BYTE := 1;
	nVersion:	E_ECODRY_VERSION;
	
	// Register Addresses. See M_UserConfigure().
	aAddr:		ARRAY [1..8] OF INT := [0, 0, 0, 0, 0, 0, 0, 0];
	aWords:		ARRAY [1..8] OF INT := [0, 0, 0, 0, 0, 0, 0, 0];
	
END_STRUCT
END_TYPE

// DUTs/Structures/Pumps/T_CRYO_PUMP_MODBUS_CTRL
TYPE T_CRYO_PUMP_MODBUS_CTRL EXTENDS T_CRYO_PUMP_BASE_CTRL:
STRUCT
	nCmdType:	DINT	:= E_MODBUS_CMD_TYPE.READ;	// Command type; 0-Read, 1-Write
	nRegister:	DINT;								// Command register
	nWords:		DINT	:= 1;						// Number of words
	nValue:		DINT;								// Parameter value
END_STRUCT
END_TYPE

// DUTs/Structures/Pumps/T_CRYO_PUMP_MODBUS_STAT
TYPE T_CRYO_PUMP_MODBUS_STAT EXTENDS T_CRYO_PUMP_BASE_STAT:
STRUCT
	nInputBuffer: 			ARRAY [0..300] OF BYTE;	// Binary data read from ECODRY
	
	lrFreqRef:				LREAL;	// Frequency Reference 0x0040
	lrOutFreq:				LREAL;	// Output Frequency 0x0041
//	lrOutCurrent:			LREAL;	// Output Current 0x0042
	lrOutVoltRef:			LREAL;	// Output Voltage Reference 0x0045
//	lrDcBusVolt:			LREAL;	// DC Bus Voltage 0x0046
	lrOutPower:				LREAL;	// Output Power 0x0047
//	lrTemperature:			LREAL;	// Heatsink Temperature 0x0068

	nSwFlash:				UINT;	// Software No. (Flash) 0x004D
	nSwRom:					UINT;	// Software No. (ROM) 0x005B
	nOpTime:				UINT;	// Accumulated Operation Time 0x004C
	nNumRunCmd:				UINT;	// Number of Run Commands 0x0075
	nFanOpTime:				UINT;	// Cooling Fan Operation Time  0x0067
	
	nServiceHours:			UINT;	// Service Hours 0x0667
	nNumPumpDowns:			UINT;	// Pump-down Cycles after Service 0x0669
	nDaysUntilService:		UINT;	// Days before Service 0x066C

END_STRUCT
END_TYPE

// DUTs/Structures/Pumps/T_CRYO_PUMP_MVP030_CFG
TYPE T_CRYO_PUMP_MVP030_CFG EXTENDS T_CRYO_PUMP_SERIAL_CFG:
STRUCT
// MVP030 specific command configuration.
// Pfeiffer Vacuum protocol for RS-485 interface.
// Assumed RS-485 device ID=1 (001) !!!

	// Definition of commands
	C_CMD_NONE:				STRING(16) := '';
	C_CMD_sCtrlViaInt:		STRING(16) := '0011006003001';	// Control via DIO
	C_CMD_sFwVersion:		STRING(16) := '0010031202=?';
	C_CMD_sHwVersion:		STRING(16) := '0010035402=?';
	C_CMD_nNominalSpeed:	STRING(16) := '0010039902=?';
	
	C_CMD_bON:				STRING(16) := '0010001002=?';
	C_CMD_nCtrlMode:		STRING(16) := '0010006002=?';
	C_CMD_sErrorCode:		STRING(16) := '0010030302=?';
	C_CMD_nMotorCurr:		STRING(16) := '0010031002=?';
	C_CMD_nPumpHours:		STRING(16) := '0010031102=?';
	C_CMD_nMotorVolt:		STRING(16) := '0010031302=?';
	C_CMD_nElecPower:		STRING(16) := '0010031602=?';
	C_CMD_nPumpTemp:		STRING(16) := '0010033002=?';
	C_CMD_nPumpSpeed:		STRING(16) := '0010039802=?';
	
	C_CMD_sID000:			STRING(16) := '0001079706000001';	// Change all IDs to 1

END_STRUCT
END_TYPE

// DUTs/Structures/Pumps/T_CRYO_PUMP_MVP030_STAT
TYPE T_CRYO_PUMP_MVP030_STAT EXTENDS T_CRYO_PUMP_BASE_STAT :
STRUCT

(*
Type:
0 - old bool: 0=FALSE, NOT 0 = TRUE.
1 - UDINT
2 - REAL * 100 (with leading zeros), e.g. 001571 corresponds with 15.71
4 - STRING (6)
7 - UINT (000 to 999)

INIT commands
312 Fw version Firmware version electronic drive unit 4 R
354 HW Version Hardware version electronic drive unit 4 R
399 NominalSpd Nominal rotation speed (rpm) 1 R rpm 0 999999

STATUS commands
010 Pumpg-Statn Pump 0 = off 1 = on 0 RW 0 1 0 x
060 CtrlViaInt Operation of the interface 
	1 = remote
	2 = RS-485
	4 = PV.can
	32 = Keys on the front panel

303 Error code Error code 4 R
	Err098 Internal communication error between interface board and drive
	Err117 Vacuum pump excess temperature (> 90 °C)
	Err174 Vacuum pump blocked
	Wrn117 High temperature vacuum pump (> 75 °C)

310 DrvCurrent Drive current 2 R A 0 9999.99
311 OpHrsPump Operating hours pump 1 R h 0 65535
313 DrvVoltage Drive voltage 2 R V 0 9999.99
316 *** DrvPower Drive power 1 R W 0 999999
330 TempPump Pump temperature 1 R °C 0 999999
398 ActualSpd Actual rotation speed (rpm) 1 R rpm 0 999999

*)

// INIT commands
	sFwVersion:		STRING(8);
	sHwVersion:		STRING(8);

// STATUS commands
	sFailureCode:	STRING(8) := 'OK';
	bTargetSpeed:	BOOL;		// Target Speed Reached
	nNominalSpeed:	DINT;		// [rpm] Nominal Pump Speed
	lrMotorVolt:	LREAL;		// Pump Motor Voltage [V]

	
	bFailure:		BOOL := FALSE;	// Err of Wrn (see cmd 303)
END_STRUCT
END_TYPE

// DUTs/Structures/Pumps/T_CRYO_PUMP_SERIAL_CFG
TYPE T_CRYO_PUMP_SERIAL_CFG EXTENDS T_CRYO_PUMP_BASE_CFG:
STRUCT
	//
	// List of INIT commands.
	//
	cmdList_Init:	ARRAY [1..8] OF T_CRYO_PUMP_CMD;

	//
	//	List of READ (and WRITE) commands.
	// NOTE: Monitoring loop stops on first cmd = ''.
	//
	cmdList_Read:	ARRAY [1..16] OF T_CRYO_PUMP_CMD;

END_STRUCT
END_TYPE

// DUTs/Structures/Sensors/T_CRYO_IOLINK_SENSOR_STATUS
TYPE T_CRYO_IOLINK_SENSOR_STATUS :
STRUCT
	bInRange:			BOOL;
	bUnderrange:		BOOL;
	bOverrange:			BOOL;
	bError:				BOOL;
	bValid:				BOOL;
	
	lrValue:			LREAL;		// Reading in UU
	
	sUnits:				STRING(16);
	sType:				STRING(32);	// Sensor type, e.g. 'Flow' or 'Temperature'.
	sStatus:			STRING	:= 'OK';

END_STRUCT
END_TYPE

// DUTs/Structures/Sensors/T_CRYO_PRESSURE_STATUS
TYPE T_CRYO_PRESSURE_STATUS :
STRUCT
	bInRange:		BOOL	:= FALSE;
	bValid:			BOOL	:= FALSE;
	bWarningSens1:	BOOL	:= TRUE;
	bWarningSens2:	BOOL	:= TRUE;
	bInVacuum:		BOOL	:= FALSE;
	bVacuumGood:	BOOL	:= FALSE;
	lrPressure:		LREAL;	// Pressure [mbar]
END_STRUCT
END_TYPE

// DUTs/Structures/Sensors/T_CRYO_PRESSURE_VOTE_STATUS
TYPE T_CRYO_PRESSURE_VOTE_STATUS :
STRUCT
	bSimulated:		BOOL;				// Flag indicating if the value is simulated.
	lrSimPressure:	LREAL;				// Simulated pressure value [mbar]

	bValid:			BOOL	:= FALSE;	// Flag indicating if the value is valid.
	lrPressure:		LREAL;				// Calculated Pressure [mbar]
	sStatus:		STRING;				// Status string

	// Flags indicating warnings for each connected sensor.
	// Only connected sensors can have warnings!!!
	bWarnSens1:		BOOL	:= TRUE;
	bWarnSens2:		BOOL	:= TRUE;
	bWarnSens3:		BOOL	:= TRUE;
	bWarnSens4:		BOOL	:= TRUE;
	bWarnSens5:		BOOL	:= TRUE;

	// Flags for each sensor indicating if it is connected.
	bConnSens1:		BOOL	:= FALSE;
	bConnSens2:		BOOL	:= FALSE;
	bConnSens3:		BOOL	:= FALSE;
	bConnSens4:		BOOL	:= FALSE;
	bConnSens5:		BOOL	:= FALSE;
END_STRUCT
END_TYPE

// DUTs/Structures/Sensors/T_CRYO_PT100_OHM2C_REC
TYPE T_CRYO_PT100_OHM2C_REC :
STRUCT
	celsius:	LREAL;	// Temperature in celsius [C]
	ohm:		LREAL;	// Resistance in [Ohm]
END_STRUCT
END_TYPE

// DUTs/Structures/Sensors/T_CRYO_SBG232_STAT
TYPE T_CRYO_SBG232_STAT :
STRUCT
	bConfigured:	BOOL;
	sName:			STRING;
	sStatus:		STRING	:= 'OK';
	
	flow:	T_CRYO_IOLINK_SENSOR_STATUS;	// Flow status
	temp:	T_CRYO_IOLINK_SENSOR_STATUS;	// Temperature status
END_STRUCT
END_TYPE

// DUTs/Structures/Sensors/T_CRYO_SENSOR_STATUS
TYPE T_CRYO_SENSOR_STATUS :
STRUCT
	//
	// Status coming from the analog input terminal.
	// This is nothing to do with the sensor, i.e. the reading can be
	// inside the input terminal measuring range but still it might
	// not be inside the sensor measuring range!
	//
	bInputUnder:		BOOL;
	bInputOver:			BOOL;
	bInputError:		BOOL;
	bInputToggle:		BOOL;
	bInputValid:		BOOL;
	bInputActive:		BOOL	:= FALSE;
	nRawValue:			INT;

	// Calculated status of the sensor
	bError:				BOOL;
	bValid:				BOOL;

END_STRUCT
END_TYPE

// DUTs/Structures/Sensors/T_CRYO_SENSOR_STATUS_PRESS
TYPE T_CRYO_SENSOR_STATUS_PRESS EXTENDS T_CRYO_SENSOR_STATUS :
STRUCT
	nType:		E_CRYO_SENSOR_TYPE_PRESS;

	// Measured and calculated values
	lrVoltage:		LREAL;	// Voltage [V]
	lrPressure:		LREAL;	// Pressure [mbar]

	// Status coming from the user evaluation.
	// These flags indicate if the reading is outside the sensor operational range.
	// Therefore, the voltage might be correctly measured but
	// the pressure is outside what the sensor can measure.	
	bValueInRange:		BOOL;	// Flag if reading is inside SENSOR(!) range
	bValueOverrange:	BOOL;	// Flag if reading is outside SENSOR(!) range
	bValueUnderrange:	BOOL;	// Flag if reading is outside SENSOR(!) range

END_STRUCT
END_TYPE

// DUTs/Structures/Sensors/T_CRYO_SENSOR_STATUS_TEMP
TYPE T_CRYO_SENSOR_STATUS_TEMP EXTENDS T_CRYO_SENSOR_STATUS :
STRUCT
	nType:		E_CRYO_SENSOR_TYPE_TEMP;
	
	lrRamp:		LREAL;	// Temperature ramp [deg/min]
	lrTempC:	LREAL;	// Temperature in deg C
	lrTempK:	LREAL;	// Temperature in deg K
END_STRUCT
END_TYPE

// DUTs/Structures/Sensors/T_CRYO_TEMPERATURE_STATUS
TYPE T_CRYO_TEMPERATURE_STATUS :
STRUCT
	bSimulated:		BOOL;				// Flag indicating if the value is simulated.
	lrSimTempK:		LREAL;				// Simulated temperature value in [K].

	bInRange:		BOOL	:= FALSE;
	bValid:			BOOL	:= FALSE;
	bWarningSens1:	BOOL	:= TRUE;
	bWarningSens2:	BOOL	:= TRUE;
	lrRamp:			LREAL;				// Temperature ramp [deg/min]
	lrTempC:		LREAL;				// Temp [deg C]
	lrTempK:		LREAL;				// Temp [deg K]
END_STRUCT
END_TYPE

// DUTs/Structures/Subsystems/Evacuation/T_CRYO_EVAC_CFG
TYPE T_CRYO_EVAC_CFG :
STRUCT
	nPressGaugeType1:	E_CRYO_SENSOR_TYPE_PRESS := E_CRYO_SENSOR_TYPE_PRESS.PKR_360;
	nPressGaugeType2:	E_CRYO_SENSOR_TYPE_PRESS := E_CRYO_SENSOR_TYPE_PRESS.PKR_360;

	bPressSimulation:	BOOL := FALSE;	// Flag is pre-vacuum pressure is simulated.

	lrThld_Prevac:					LREAL := 0.005;	// Prevacuum pressure threshold
	lrThld_PrevacHigh:				LREAL := 5.0;	// Prevacuum pressure too high threshold
	// Cryo pressure threshold for safe Turbo Pump start
	lrThld_TP_SafeStartPressure:	LREAL := 0.01;	
	// Cryo pressure threshold for safe Valve opening
	lrThld_Valve_SafeOpenPressure:	LREAL := 0.1;	
	
	tDelay:		TIME := T#3S;	// Time delay before stopping Turbo Pump
END_STRUCT
END_TYPE

// DUTs/Structures/Subsystems/Evacuation/T_CRYO_EVAC_CFG_50000
TYPE T_CRYO_EVAC_CFG_50000 :
STRUCT
	// Pressure sensor gauge types
	nType_VAG1:		E_CRYO_SENSOR_TYPE_PRESS := E_CRYO_SENSOR_TYPE_PRESS.PKR_360;
	nType_VAG2:		E_CRYO_SENSOR_TYPE_PRESS := E_CRYO_SENSOR_TYPE_PRESS.PKR_360;
	nType_VAG3:		E_CRYO_SENSOR_TYPE_PRESS := E_CRYO_SENSOR_TYPE_PRESS.PKR_360;
	nType_VAGF1:	E_CRYO_SENSOR_TYPE_PRESS := E_CRYO_SENSOR_TYPE_PRESS.PKR_360;
	nType_VAGF2:	E_CRYO_SENSOR_TYPE_PRESS := E_CRYO_SENSOR_TYPE_PRESS.PKR_360;
	nType_VAGG1:	E_CRYO_SENSOR_TYPE_PRESS := E_CRYO_SENSOR_TYPE_PRESS.PKR_360;
	nType_VAGG2:	E_CRYO_SENSOR_TYPE_PRESS := E_CRYO_SENSOR_TYPE_PRESS.PKR_360;

	// Flag is pressures are simulated.
	// TODO: Define individual flags for each sensor.
	bPressSimulation:	BOOL := FALSE;	

	lrThld_Prevac:			LREAL := 0.1;	// Prevacuum pressure threshold [mbar] 
	lrThld_PrevacHigh:		LREAL := 5.0;	// Prevacuum pressure too high threshold [mbar]
	lrThld_Vacuum:			LREAL := 0.0001;// At this Cryo pressure evacuation has started [mbar]
	
	tDelay:		TIME := T#3S;	// Delay after closing all valves before stopping Pumps
END_STRUCT
END_TYPE

// DUTs/Structures/Subsystems/Evacuation/T_CRYO_EVAC_CTRL
TYPE T_CRYO_EVAC_CTRL :
STRUCT
	bEnable_RP:		BOOL := FALSE;
	bEnable_TP:		BOOL := FALSE;
	bEnable_Valve:	BOOL := FALSE;
END_STRUCT
END_TYPE

// DUTs/Structures/Subsystems/Evacuation/T_CRYO_EVAC_CTRL_50000
TYPE T_CRYO_EVAC_CTRL_50000 :
STRUCT
	// Flags for control of pumps.
	// Seeting the flag to TRUE  will start the pump.
	// Seeting the flag to FALSE will stop  the pump.
	bEnable_PVP:	BOOL := FALSE;	// Prevacuum pump
	bEnable_TMP:	BOOL := FALSE;	// Turbo molecular pump
	
	// Flags for control of valves
	// Seeting the flag to TRUE  will open  the valve.
	// Seeting the flag to FALSE will close the valve.
	bEnable_PVV1:	BOOL := FALSE;
	bEnable_PVV2:	BOOL := FALSE;
	bEnable_PVV3:	BOOL := FALSE;
	bEnable_PVV4:	BOOL := FALSE;
	bEnable_GBV:	BOOL := FALSE;
	
END_STRUCT
END_TYPE

// DUTs/Structures/Subsystems/Evacuation/T_CRYO_EVAC_STAT
TYPE T_CRYO_EVAC_STAT :
STRUCT
	bEnabled:		BOOL := FALSE;	// Controller active while bEnable is TRUE
	bConfigured:	BOOL := FALSE;	// Flag if controller has been configured.
	bError:			BOOL;			// Flag if controller is OK
	bActive:		BOOL;			// Flag if controller is ACTIVE
	bEmergency:		BOOL := FALSE;	// Flag if there was Emergency valve closure
	bRootPumpON:	BOOL;			// Flag if Root Pump is running
	bTurboPumpON:	BOOL;			// Flag if Turbo Pump is running
	bValveOpen:		BOOL;			// Flag if Evacuation Valve is open
	bValveAfterTP:	BOOL := FALSE;	// Flag if Evacuation Valve should open after TP has started

	// Generic controller OK flag.
	// Used for problems other than from the actuator.
	// This flag is used for problems coming from controllers
	// that extend the functionality of FB_CRYO_BIN_CTRL.
	bCtrlOK:	BOOL := TRUE;		

	nCycleCounter:	UDINT := 0;
	nState:			E_CRYO_EVAC_STATE	:= E_CRYO_EVAC_STATE.NONE;
	
	sErrorText:		STRING(64);		// Error as text
	sState:			STRING(64);		// State as text
	sStatus:		STRING(64);		// Status as text
END_STRUCT
END_TYPE

// DUTs/Structures/Subsystems/Evacuation/T_CRYO_EVAC_STAT_50000
TYPE T_CRYO_EVAC_STAT_50000 :
STRUCT
	bEnabled:		BOOL := FALSE;	// Controller active while bEnable is TRUE
	bConfigured:	BOOL := FALSE;	// Flag if controller has been configured.
	bError:			BOOL;			// Flag if controller is OK
	bActive:		BOOL;			// Flag if controller is ACTIVE
	bEmergency:		BOOL := FALSE;	// Flag if there was Emergency valve closure
	bRootPumpON:	BOOL;			// Flag if Root Pump is running
	bTurboPumpON:	BOOL;			// Flag if Turbo Pump is running

	// Generic controller OK flag.
	// Used for problems other than from the actuator.
	// This flag is used for problems coming from controllers
	// that extend the functionality of FB_CRYO_BIN_CTRL.
	bCtrlOK:	BOOL := TRUE;		

	nCycleCounter:	UDINT := 0;
	nState:			E_CRYO_EVAC_STATE_50000	:= E_CRYO_EVAC_STATE_50000.NONE;
	
	sErrorText:		STRING(64);		// Error as text
	sState:			STRING(64);		// State as text
	sStatus:		STRING(64);		// Status as text
END_STRUCT
END_TYPE

// DUTs/Structures/Subsystems/Evacuation/T_CRYO_EVAC_SYS_INPUT
// NOTE: Not used yet !!!
// Should replace input parameters of FB_CRYO_EVACUATION_SYSTEM.
// Should be set with NEW method FB_CRYO_CTRL::M_SetEvacSystemInputData().
TYPE T_CRYO_EVAC_SYS_INPUT :
STRUCT
	//
	// System configuration
	//
	// Time between closing Vac valve and Switching OFF the vac Pump [ms]
	nTime_DeltaTValve:		UDINT;	
	// Time [ms] to run Turbo Pump to consider vacuum is good (useful when cryostat is cold)
	nTime_TurboPump:		UDINT;	

	lrPress_Atm:			LREAL;	// Atmospheric pressure limit   [mbar]

	lrTemp_Precooled:		LREAL;	// Precooled temperature limit [K]
	lrTemp_Warm:			LREAL;	// Warm      temperature limit [K]

	//
	// System configuration
	//
	lrTemp_Cryo:			T_CRYO_TEMPERATURE_STATUS;	// Cold Bench temperature	
	lrPressure_Cryo:		T_CRYO_PRESSURE_STATUS;		// Cryostat Pressure
	lrPressure_Evac:		T_CRYO_PRESSURE_STATUS;		// Evacuation Pressure
	bRepressValveOpen:		BOOL;	// Repressure Valve Open flag
	bRepressValveOK:		BOOL;	// Repressure Valve OK flag
END_STRUCT
END_TYPE

// DUTs/Structures/Subsystems/Evacuation/T_CRYO_EVACUATION_SYSTEM_STATUS
TYPE T_CRYO_EVACUATION_SYSTEM_STATUS :
STRUCT
	bDone:			BOOL;			// Flag if controller is OK
	bBusy:			BOOL;			// Flag if controller is BUSY
	bEnabled:		BOOL := FALSE;	// Controller active while bEnable is TRUE
	bError:			BOOL;			// Flag if controller is OK
	bActive:		BOOL;			// Flag if controller is ACTIVE
	bEmergency:		BOOL := FALSE;	// Flag if there was Emergency valve closure
	bRootPumpON:	BOOL;			// Flag if Root Pump is running
	bTurboPumpON:	BOOL;			// Flag if Turbo Pump is running
	bTurboPump10min:BOOL;			// Flag if Turbo Pump has been running for more than 10 min
	bValveOpen:		BOOL;			// Flag if Evacuation Valve is open

	// Generic controller OK flag.
	// Used for problems other than from the actuator.
	// This flag is used for problems coming from controllers
	// that extend the functionality of FB_CRYO_BIN_CTRL.
	bCtrlOK:	BOOL := TRUE;		

	nCycleCounter:	UDINT := 0;
	nLastCommand:	E_CRYO_BIN_ACT_CMD	:= E_CRYO_BIN_ACT_CMD.NONE;	// Command
	nState:			E_CRYO_EVAC_SYS_STATE	:= E_CRYO_EVAC_SYS_STATE.NONE;
	
	sState:			STRING(64);		// State as text
	sStatus:		STRING(64);		// Status as text
END_STRUCT
END_TYPE

// DUTs/Structures/System/T_CRYO_CFG
TYPE T_CRYO_CFG :
STRUCT
	lrTemp_Precooled:		LREAL := 110.0;	// Precooled temperature limit [K]
	lrTemp_Cold:			LREAL :=  80.0;	// Cool      temperature limit [K]
	lrTemp_Warm:			LREAL := 283.15;// Warm      temperature limit [K] = 10 C
	
	// Delat-T SetPoint between Detector and Coldbench during WarmUp
	lrTemp_DeltaDet_Bench_Low:	LREAL	:= 10.0;
	// Delat-T SetPoint between Detector and Coldbench during WarmUp	
	lrTemp_DeltaDet_Bench_High:	LREAL	:= 5.0;		

	lrTemp_LN2ValveOpen:	LREAL := 91.27;		// Open  valve if temperature above this value [K]
	lrTemp_LN2ValveClose:	LREAL := 79.148;	// Close valve if temperature below this value [K]

	lrPress_Atm:			LREAL := 700.0;		// Atmospheric pressure limit   [mbar]
	lrPress_InVac:			LREAL := 10.0E-1;	// In vacuum limit   [mbar]
	lrPress_GoodVac:		LREAL := 10.0E-4;	// Good Vacuum limit [mbar]
	
	
	// Time between closing Vac valve and Switching OFF the vac Pump [ms]
	nTime_DeltaTValve:		UDINT := 2000;	
	// Vacuum Pump Settling Time [ms]
	nTime_VacPumpSettling:	UDINT := 1000;	
	// 10 min (600000ms) run of Turbo Pump to consider vac is good (useful when cryostat is cold)
	nTime_TurboPump:		UDINT := 600000;	
	
	//
	// Lakeshore 340 configuration
	//
	LS_CTRL_MODE:			INT		:= 2;		// Remote without local lock
	
	// Warm
	LS_W_PID_A_P:			UINT	:= 10;		// Warm state P controler value
	LS_W_PID_A_I:			UINT	:= 50;		// Warm state I controler value
	LS_W_PID_A_D:			UINT	:= 12;		// Warm state D controler value
	LS_W_Heater_Range:		UINT	:= 4;		// Warm Resistance power range
	LS_W_CTRL_RAMP:			LREAL	:= 1.0;		// Warm-up delta-T Kelvin per minutes
	LS_W_SETPOINT_A:		LREAL	:= 293.15;	// 20 Deg Celcius

	// Cold
	LS_C_PID_A_P:			UINT	:= 50;		// Cold state P controler value
	LS_C_PID_A_I:			UINT	:= 71;		// Cold state I controler value
	LS_C_PID_A_D:			UINT	:= 10;		// Cold state D controler value
	LS_C_Heater_Range:		UINT	:= 4;		// Cold Resistance power range
	LS_C_CTRL_RAMP:			LREAL	:= 0.0;		// Cooldown/Cooling delta-T Kelvin per minutes
	LS_C_SETPOINT_A:		LREAL	:= 40.0;	// -193,15 Deg Celcius

END_STRUCT
END_TYPE

// DUTs/Structures/System/T_CRYO_CTRL
TYPE T_CRYO_CTRL :
STRUCT
	bExecute:	BOOL := FALSE;
	nCommand:	E_CRYO_CTRL_CMD := E_CRYO_CTRL_CMD.NONE;
	
	bReset:		BOOL := FALSE;		// RESET Command

	bEnable_Evac:		BOOL := FALSE;
	bEnable_Heater:		BOOL := FALSE;
	bEnable_Precool:	BOOL := FALSE;
	bEnable_Cool:		BOOL := FALSE;
	bEnable_Warmup:		BOOL := FALSE;
	bEnable_CCC:		BOOL := FALSE;
	bEnable_RepressSys:	BOOL := FALSE;
	bEnable_RepressCtrl:BOOL := FALSE;

	// Safe flags
	bSafe_Precool:		BOOL := FALSE;
	bSafe_Cooling:		BOOL := FALSE;
	bSafe_Warmup:		BOOL := FALSE;
	bSafe_Repress:		BOOL := FALSE;
	
	// Ignore underrange flags.
	// We know that the ColdBench PT100 is broken and gives -200 C.
	bIgnoreUnderrange_ColdBench:	BOOL := FALSE;
	
	// Lakeshore related control parameters
	bLS_UpdateSETP:		BOOL := FALSE;	// If TRUE, this flag will trigger Lakeshore SETP.
	lrLS_SETP:			LREAL := 40.0;	// New SETP
	lrLS_RAMP:			LREAL := 0.5;	// RAMP [K/min]
	
END_STRUCT
END_TYPE

// DUTs/Structures/System/T_CRYO_LOG
// Last ten system logs
TYPE T_CRYO_LOG :
STRUCT
	// This could have been done much simpler as:
	// 	sLog: ARRAY [0..9] OF STRING(80);
	// However, this would make it hard to view individual strings
	// with OPC UA Clients.
	// That's why we use 'ptrLog[0..9]' to scroll through the strings.
	// See M_Configure() for how pointers are set.
	
	s0:		STRING(80);
	s1:		STRING(80);
	s2:		STRING(80);
	s3:		STRING(80);
	s4:		STRING(80);
	s5:		STRING(80);
	s6:		STRING(80);
	s7:		STRING(80);
	s8:		STRING(80);
	s9:		STRING(80);
END_STRUCT
END_TYPE

// DUTs/Structures/System/T_CRYO_STAT
TYPE T_CRYO_STAT :
STRUCT
	bConfigured:	BOOL := FALSE;

	bDone:			BOOL;			// Flag if controller is OK
	bBusy:			BOOL;			// Flag if controller is BUSY
	bError:			BOOL;			// Flag if controller is OK
	bActive:		BOOL;			// Flag if controller is ACTIVE
	// Generic controller OK flag.
	// Used for problems other than from the actuator.
	// This flag is used for problems coming from controllers
	// that extend the functionality of FB_CRYO_BIN_CTRL.
	bCtrlOK:		BOOL := TRUE;		

	bInVacuum:		BOOL := FALSE;		
	bGoodVacuum:	BOOL := FALSE;		

	bHighestTempValid:	BOOL := FALSE;	// Highest temperature Valid flag
	bLowestTempValid:	BOOL := FALSE;	// Lowest temperature Valid flag
	bDiffTempValid:		BOOL := FALSE;	// TRUE if Temperature difference is Valid

	lrHighestTempK:	LREAL;	// Highest temperature [K] in Cryostat
	lrLowestTempK:	LREAL;	// Lowest temperature [K] in Cryostat
	lrDiffTempK:	LREAL;	// Temperature difference (DET -Lowest temperature) [K]
	lrLS_Power:		LREAL;	// Lakeshore Power Output [%]
	
	nCycleCounter:	UDINT := 0;
	nLastCommand:	E_CRYO_CTRL_CMD 	:= E_CRYO_CTRL_CMD.NONE;
	nState:			E_CRYO_CTRL_STATE	:= E_CRYO_CTRL_STATE.NONE;
	
	
	sState:			STRING(64);		// State as text

END_STRUCT
END_TYPE

// POUs/Actuators/FB_CRYO_ACTUATOR_CMD
FUNCTION_BLOCK FB_CRYO_ACTUATOR_CMD
VAR_INPUT
	in_bEnable:		BOOL;			// External ON/OFF command
	in_bInterlock:	BOOL := FALSE;	// External Interlock
END_VAR
VAR_OUTPUT
	out_bEnable:	BOOL := FALSE;	// Resulting command
END_VAR
VAR
	bAutoMode:		BOOL := TRUE;	// AUTO=true, MANUAL=false
	bEngMode:		BOOL := FALSE;	// Commissioning/Engineering mode. Ignores interlocks
	
	// Disable/enable manual control buttons
	bDisableBtnOn:	BOOL := FALSE;
	bDisableBtnOff:	BOOL := FALSE;

	// ON/OFF command permissions
	bPermitOn:		BOOL := TRUE;
	bPermitOff:		BOOL := TRUE;
	
	// Handling of Manual commands
	bManualCmd:		BOOL := FALSE;
	bManualExecute:	BOOL := FALSE;
	
	// Reset interlocks (if possible)
	bReset:			BOOL := FALSE;
END_VAR

IF bAutoMode THEN
	// Simplest case, no restrictions.
	out_bEnable	:= in_bEnable;
	// Disable Manual control buttons
	bDisableBtnOn	:= TRUE;
	bDisableBtnOff	:= TRUE;
ELSIF bEngMode	THEN
	// No restrictions, no safety !!!
	// User responsible for damage caused by wrong/dangerous commands.
	IF bManualExecute THEN
		// Assign user command to the output without any checks !!!
		out_bEnable		:= bManualCmd;
		// Clear command trigger
		bManualExecute	:= FALSE;
	END_IF
	// Enable Manual control buttons
	bDisableBtnOn	:= FALSE;
	bDisableBtnOff	:= FALSE;
ELSIF NOT bAutoMode	THEN
	//
	// Manual mode.
	//
	// Only permitted commands can be executed.
	IF bManualExecute THEN
		// Execute only permitted commands.
		IF	(bManualCmd = TRUE   AND  bPermitOn)  OR
			(bManualCmd = FALSE  AND  bPermitOff) 	THEN
			// Assign user command to the output.
			out_bEnable		:= bManualCmd;
		END_IF
		// Clear command trigger
		bManualExecute	:= FALSE;
	ELSIF in_bInterlock THEN 
		// Interlock active
		IF bPermitOn AND bPermitOff THEN
			// Enable Manual control of both ON&OFF buttons
			bDisableBtnOn	:= FALSE;
			bDisableBtnOff	:= FALSE;
		ELSIF bPermitOn THEN
			// Manual Mode and only ON is permitted.
			out_bEnable		:= TRUE;
			// Enable Manual control ON button
			bDisableBtnOn	:= FALSE;
			bDisableBtnOff	:= TRUE;
		ELSIF bPermitOff THEN
			// Manual Mode and only OFF is permitted.
			out_bEnable		:= FALSE;
			// Enable Manual control OFF button
			bDisableBtnOn	:= TRUE;
			bDisableBtnOff	:= FALSE;
		END_IF
	ELSIF NOT in_bInterlock THEN
		// Enable/Disable Manual control buttons
		bDisableBtnOn	:= NOT bPermitOn;
		bDisableBtnOff	:= NOT bPermitOFF;
	END_IF
END_IF

METHOD M_SetPermissionOff
VAR_INPUT
	in_bPermit:	BOOL;
END_VAR
bPermitOff	:= in_bPermit;
END_METHOD

METHOD M_SetPermissionOn
VAR_INPUT
	in_bPermit:	BOOL;
END_VAR
bPermitOn	:= in_bPermit;
END_METHOD

METHOD M_SetPermissions
VAR_INPUT
	in_bPermitOn:	BOOL;
	in_bPermitOff:	BOOL;
END_VAR
bPermitOn	:= in_bPermitOn;
bPermitOff	:= in_bPermitOff;
END_METHOD

END_FUNCTION_BLOCK

// POUs/Actuators/FB_CRYO_BIN_ACT
FUNCTION_BLOCK FB_CRYO_BIN_ACT
VAR_INPUT
	in_nFeedback:		E_CRYO_BIN_ACT_FEEDBACK := E_CRYO_BIN_ACT_FEEDBACK.ON_ONLY;	// Feedback configuration.
	in_nTimeout:		UDINT := 10000;	// Timeout for switching on/off [ms]. Default 10000.
	in_bActiveLowCtrl:	BOOL := FALSE;	// Active Low for Control output
	in_bActiveLowStat:	BOOL := FALSE;	// Active Low for Status signals, i.e. feedback
	in_nCommand:		E_CRYO_BIN_ACT_CMD	:= E_CRYO_BIN_ACT_CMD.NONE;	// Command
	in_bExecute:		BOOL := FALSE;	// Execute trigger
END_VAR
VAR
	{attribute 'OPC.UA.DA' := '0'}
	i_nCouplerState	AT%I*:	UINT;		// Terminal state. Should be 8, i.e. OP.
	{attribute 'OPC.UA.DA' := '0'}
	i_bON			AT%I*:	BOOL;		// Feedback for ON
	{attribute 'OPC.UA.DA' := '0'}
	i_bOFF			AT%I*:	BOOL;		// Feedback for OFF
	
	{attribute 'OPC.UA.DA' := '0'}
	q_bCtrl			AT%Q*:	BOOL;		// Control output signal
	
	stat:		T_CRYO_BIN_ACT_STATUS;

	
	{attribute 'OPC.UA.DA' := '0'}
	timer:		TON;		// Timer for commands
	{attribute 'OPC.UA.DA' := '0'}
	trigCMD:	R_TRIG;		// Trigger for new command
	
	{attribute 'OPC.UA.DA' := '0'}
	nCommand:	E_CRYO_BIN_ACT_CMD	:= E_CRYO_BIN_ACT_CMD.NONE;	// Command

END_VAR

// Get the feedback
M_GetFeedback();

// Check for new command
trigCMD(CLK:=in_bExecute);
IF trigCMD.Q THEN
	nCommand			:= in_nCommand;
	stat.nLastCommand	:= in_nCommand;
ELSE
	nCommand		:= E_CRYO_BIN_ACT_CMD.NONE;
END_IF

// If the system is not operational, this is an error.
IF i_nCouplerState <> 8 THEN
	stat.nState	:= E_CRYO_BIN_ACT_STATE.ERROR;
	stat.sState	:= 'ERROR: System not OPERATIONAL';
	M_SetStatus(stat.nState);	
END_IF

CASE stat.nState OF
	/////////////////////////////////
	E_CRYO_BIN_ACT_STATE.NONE:
	/////////////////////////////////
	//
	// Determine the initial state based on the feedback
	IF stat.bON	THEN
		stat.nState	:= E_CRYO_BIN_ACT_STATE.ON;
	ELSIF stat.bOFF	THEN
		stat.nState	:= E_CRYO_BIN_ACT_STATE.OFF;
	ELSE
		stat.nState	:= E_CRYO_BIN_ACT_STATE.ERROR;
		stat.sState	:= 'ERROR';
	END_IF
	M_SetStatus(stat.nState);	
	RETURN;
	

	/////////////////////////////////
	E_CRYO_BIN_ACT_STATE.OFF:
	/////////////////////////////////
	//
	IF	stat.bON  OR  
		stat.bError	THEN
		// This should never happen in state OFF
		stat.nState	:= E_CRYO_BIN_ACT_STATE.ERROR;
		stat.sState	:= 'ERROR: Lost ON state.';
		M_SetStatus(stat.nState);	
	ELSE
		// Check for command to go ON
		IF nCommand = E_CRYO_BIN_ACT_CMD.ON THEN
			// Start the timer
			timer(IN:=FALSE);
			timer(IN:=TRUE, PT:=UDINT_TO_TIME(in_nTimeout));
			// Activate the output
			M_SetCtrlOutput(TRUE);
			// Goto SWITCHING_ON state
			stat.nState	:= E_CRYO_BIN_ACT_STATE.SWITCHING_ON;
			M_SetStatus(stat.nState);	
		END_IF
	END_IF
	RETURN;
	
	
	/////////////////////////////////
	E_CRYO_BIN_ACT_STATE.SWITCHING_ON:
	/////////////////////////////////
	//
	// Check for timeout
	timer(IN:=TRUE);
	IF timer.Q THEN
		// Stop the timer
		timer(IN:=FALSE);
		// Goto ERROR state
		stat.nState	:= E_CRYO_BIN_ACT_STATE.ERROR;
		stat.sState	:= 'ERROR: Timeout switching ON';
		M_SetStatus(stat.nState);	
		RETURN;
	END_IF
	
	// Check if we have reached ON state
	IF stat.bON	AND NOT stat.bOFF	THEN
		// Stop the timer
		timer(IN:=FALSE);
		// Goto ON state
		stat.nState	:= E_CRYO_BIN_ACT_STATE.ON;
		M_SetStatus(stat.nState);	
	END_IF
	RETURN;
	

	/////////////////////////////////
	E_CRYO_BIN_ACT_STATE.ON:
	/////////////////////////////////
	//
	IF	stat.bOFF  OR  
		stat.bError	THEN
		// This should never happen in state ON
		stat.nState	:= E_CRYO_BIN_ACT_STATE.ERROR;
		stat.sState	:= 'ERROR: Lost OFF state.';
		M_SetStatus(stat.nState);	
	ELSE
		// Check for command to go OFF
		IF nCommand = E_CRYO_BIN_ACT_CMD.OFF THEN
			// Start the timer
			timer(IN:=FALSE);
			timer(IN:=TRUE, PT:=UDINT_TO_TIME(in_nTimeout));
			// Deactivate the output
			M_SetCtrlOutput(FALSE);
			// Goto SWITCHING_OFF state
			stat.nState	:= E_CRYO_BIN_ACT_STATE.SWITCHING_OFF;
			M_SetStatus(stat.nState);	
		END_IF
	END_IF
	RETURN;
	
	
	//////////////////////////////////
	E_CRYO_BIN_ACT_STATE.SWITCHING_OFF:
	//////////////////////////////////
	//
	// Check for timeout
	timer(IN:=TRUE);
	IF timer.Q THEN
		// Stop the timer
		timer(IN:=FALSE);
		// Goto ERROR state
		stat.nState	:= E_CRYO_BIN_ACT_STATE.ERROR;
		stat.sState	:= 'ERROR: Timeout switching OFF';
		M_SetStatus(stat.nState);	
		RETURN;
	END_IF
	
	// Check if we have reached OFF state
	IF stat.bOFF AND NOT stat.bON	THEN
		// Stop the timer
		timer(IN:=FALSE);
		// Goto OFF state
		stat.nState	:= E_CRYO_BIN_ACT_STATE.OFF;
		M_SetStatus(stat.nState);	
	END_IF
	RETURN;
	
	/////////////////////////////////
	E_CRYO_BIN_ACT_STATE.ERROR:
	/////////////////////////////////
	//
	// Deactivate the output
	M_SetCtrlOutput(FALSE);
	
	// Check for command to go ON
	IF nCommand = E_CRYO_BIN_ACT_CMD.ON THEN
		// Start the timer
		timer(IN:=FALSE);
		timer(IN:=TRUE, PT:=UDINT_TO_TIME(in_nTimeout));
		// Activate the output
		M_SetCtrlOutput(TRUE);
		// Goto SWITCHING_ON state
		stat.nState	:= E_CRYO_BIN_ACT_STATE.SWITCHING_ON;
		M_SetStatus(stat.nState);	
	// Check for command to go OFF
	ELSIF nCommand = E_CRYO_BIN_ACT_CMD.OFF THEN
		// Start the timer
		timer(IN:=FALSE);
		timer(IN:=TRUE, PT:=UDINT_TO_TIME(in_nTimeout));
		// Deactivate the output
		M_SetCtrlOutput(FALSE);
		// Goto SWITCHING_OFF state
		stat.nState	:= E_CRYO_BIN_ACT_STATE.SWITCHING_OFF;
		M_SetStatus(stat.nState);	
	END_IF
	RETURN;

END_CASE

METHOD M_GetFeedback
VAR_INPUT
END_VAR
// Get ON/OFF status based on active low configuration
IF in_bActiveLowStat	THEN
	stat.bON	:= NOT i_bON;
	stat.bOFF	:= NOT i_bOFF;
ELSE
	stat.bON	:= i_bON;
	stat.bOFF	:= i_bOFF;
END_IF

// Check for possible feedback errors.
// Also, adjust the OFF signal, if only ON feedback exists.
IF in_nFeedback = E_CRYO_BIN_ACT_FEEDBACK.ON_AND_OFF  THEN
	// There are separate signals for ON and OFF.
	// The status is already properly assigned. Nothing more to do.
	// If both feedback signals are active, this is an error.
	(*
	IF stat.bON AND stat.bOFF	THEN
		stat.nState	:= E_CRYO_BIN_ACT_STATE.ERROR;
		stat.sState	:= 'ERROR: Both ON and OFF signals active!';
		M_SetStatus(stat.nState);	
	END_IF
	*)
	;
ELSIF in_nFeedback = E_CRYO_BIN_ACT_FEEDBACK.ON_ONLY  THEN
	// There is only a feedback signal for ON.
	// Therefore, stat.bOFF := NOT stat.bON
	stat.bOFF	:= NOT stat.bON;
END_IF
END_METHOD

METHOD M_SetCtrlOutput
VAR_INPUT
	in_bSignal:	BOOL;
END_VAR
// Set control output signal based on active low configuration
IF in_bActiveLowCtrl	THEN
	q_bCtrl	:= NOT in_bSignal;
ELSE
	q_bCtrl	:= in_bSignal;
END_IF
END_METHOD

METHOD M_SetStatus
VAR_INPUT
	nState:	E_CRYO_BIN_ACT_STATE;
END_VAR
CASE stat.nState OF
	
	E_CRYO_BIN_ACT_STATE.OFF,
	E_CRYO_BIN_ACT_STATE.ON:
	stat.bDone	:= TRUE;
	stat.bBusy	:= FALSE;
	stat.bError	:= FALSE;
	
	E_CRYO_BIN_ACT_STATE.SWITCHING_ON,
	E_CRYO_BIN_ACT_STATE.SWITCHING_OFF:
	stat.bDone	:= FALSE;
	stat.bBusy	:= TRUE;
	stat.bError	:= FALSE;
	
	E_CRYO_BIN_ACT_STATE.ERROR:
	stat.bDone	:= TRUE;
	stat.bBusy	:= FALSE;
	stat.bError	:= TRUE;
END_CASE

// Set status string
CASE stat.nState OF
	
	E_CRYO_BIN_ACT_STATE.OFF:
	stat.sState	:= 'OFF';
	
	E_CRYO_BIN_ACT_STATE.ON:
	stat.sState	:= 'ON';
	
	E_CRYO_BIN_ACT_STATE.SWITCHING_ON:
	stat.sState	:= 'SWITCHING_ON...';
	
	E_CRYO_BIN_ACT_STATE.SWITCHING_OFF:
	stat.sState	:= 'SWITCHING_OFF...';
	
	E_CRYO_BIN_ACT_STATE.ERROR:
	// Error string was set where the error was detected.
	//	stat.sState	:= 'ERROR';
	;
END_CASE
END_METHOD

END_FUNCTION_BLOCK

// POUs/Actuators/FB_CRYO_BIN_CTRL
// Binary Controller
FUNCTION_BLOCK FB_CRYO_BIN_CTRL
VAR_INPUT
	in_nFeedback:		E_CRYO_BIN_ACT_FEEDBACK := E_CRYO_BIN_ACT_FEEDBACK.ON_ONLY;	// Feedbacks
	in_nTimeout:		UDINT := 10000;	// Timeout for switching on/off [ms]. Default 10000.
	in_bActiveLowCtrl:	BOOL := FALSE;	// Active Low for Control output
	in_bActiveLowStat:	BOOL := FALSE;	// Active Low for Status signals, i.e. feedback
	in_bEnable:			BOOL := FALSE;	// Controller active while in_bEnable is TRUE
END_VAR
VAR
	
	{attribute 'OPC.UA.DA' := '1'}
	Actuator:	FB_CRYO_BIN_ACT;	// Heater, valve, etc.
	
	stat:		T_CRYO_BIN_CTRL_STATUS;


	{attribute 'OPC.UA.DA' := '0'}
	bReset:		BOOL := FALSE;		// RESET Command


	{attribute 'OPC.UA.DA' := '0'}
	timer:		TON;		// Timer for commands
	
	
END_VAR

// Increment cycle counter
stat.nCycleCounter := stat.nCycleCounter + 1;

// Execute Actuator FB on every cycle
Actuator(
	in_nFeedback		:= in_nFeedback,
	in_nTimeout			:= in_nTimeout,
	in_bActiveLowCtrl	:= in_bActiveLowCtrl,
	in_bActiveLowStat	:= in_bActiveLowStat);


CASE stat.nState OF
	/////////////////////////////////
	E_CRYO_BIN_CTRL_STATE.NONE:
	/////////////////////////////////
	//
	// This is the state on power-up.
	// Determine the initial state based on the command amd actuator state.
	IF Actuator.stat.bError  OR NOT stat.bCtrlOK	THEN
		stat.nState	:= E_CRYO_BIN_CTRL_STATE.ERROR;
	ELSIF in_bEnable  AND  Actuator.stat.bON	THEN
		stat.nState	:= E_CRYO_BIN_CTRL_STATE.ACTIVE_ON;
	ELSIF in_bEnable  AND  Actuator.stat.bOFF	THEN
		stat.nState	:= E_CRYO_BIN_CTRL_STATE.ACTIVE_OFF;
	ELSIF NOT in_bEnable  THEN
		stat.nState	:= E_CRYO_BIN_CTRL_STATE.OFF;
	END_IF
	M_SetStatus(stat.nState);	
	RETURN;
	

	/////////////////////////////////
	E_CRYO_BIN_CTRL_STATE.OFF:
	/////////////////////////////////
	//
	IF	Actuator.stat.bError	OR NOT stat.bCtrlOK	THEN
		stat.nState	:= E_CRYO_BIN_CTRL_STATE.ERROR;
	ELSIF in_bEnable  THEN
		// Activate the control loop.
		// Goto Active_Off first.
		//
		// Start the timer
		timer(IN:=FALSE);
		timer(IN:=TRUE, PT:=UDINT_TO_TIME(in_nTimeout));
		// Set next state
		stat.nState	:= E_CRYO_BIN_CTRL_STATE.ACTIVE_OFF;
	END_IF
	M_SetStatus(stat.nState);	
	RETURN;
	
	
	/////////////////////////////////
	E_CRYO_BIN_CTRL_STATE.ACTIVE_OFF:
	/////////////////////////////////
	//
	IF	Actuator.stat.bError	OR NOT stat.bCtrlOK  THEN
		stat.nState	:= E_CRYO_BIN_CTRL_STATE.ERROR;
	ELSIF NOT in_bEnable  THEN
		// Goto Off.
		//
		// Set next state
		stat.nState	:= E_CRYO_BIN_CTRL_STATE.OFF;
	ELSIF M_User_SetAction() = E_CRYO_BIN_CTRL_ACTION.ON THEN
		// Goto Active_Off.
		//
		// Start the timer
		timer(IN:=FALSE);
		timer(IN:=TRUE, PT:=UDINT_TO_TIME(in_nTimeout));
		
		// Trigger action
		Actuator(in_bExecute:=FALSE);
		Actuator(in_bExecute:=TRUE, in_nCommand:=E_CRYO_BIN_ACT_CMD.ON);
		
		// Set next state
		stat.nState	:= E_CRYO_BIN_CTRL_STATE.ACTIVE_SWITCHING_ON;
	END_IF
	M_SetStatus(stat.nState);	
	RETURN;
	
	
	//////////////////////////////////////////
	E_CRYO_BIN_CTRL_STATE.ACTIVE_SWITCHING_ON:
	//////////////////////////////////////////
	//
	// Check for timeout
	timer(IN:=TRUE);
	IF timer.Q THEN
		// Stop the timer
		timer(IN:=FALSE);
		// Goto ERROR state
		stat.nState	:= E_CRYO_BIN_CTRL_STATE.ERROR;
	ELSIF	Actuator.stat.bError	THEN
		stat.nState	:= E_CRYO_BIN_CTRL_STATE.ERROR;
	ELSIF Actuator.stat.bON THEN
		// The actuator is ON, transition completed.
		// Goto Active_On.
		stat.nState	:= E_CRYO_BIN_CTRL_STATE.ACTIVE_ON;
	END_IF
	M_SetStatus(stat.nState);	
	RETURN;
	

	/////////////////////////////////
	E_CRYO_BIN_CTRL_STATE.ACTIVE_ON:
	/////////////////////////////////
	//
	IF	Actuator.stat.bError	THEN
		stat.nState	:= E_CRYO_BIN_CTRL_STATE.ERROR;
	ELSIF	NOT in_bEnable 		OR  
			NOT stat.bCtrlOK	OR
			M_User_SetAction() = E_CRYO_BIN_CTRL_ACTION.OFF THEN
		// Goto Active_Off.
		// If NOT in_bExecute, the system will continue to complete OFF
		//
		// Start the timer
		timer(IN:=FALSE);
		timer(IN:=TRUE, PT:=UDINT_TO_TIME(in_nTimeout));
		
		// Trigger action
		Actuator(in_bExecute:=FALSE);
		Actuator(in_bExecute:=TRUE, in_nCommand:=E_CRYO_BIN_ACT_CMD.OFF);
		
		// Set next state
		stat.nState	:= E_CRYO_BIN_CTRL_STATE.ACTIVE_SWITCHING_OFF;
	END_IF
	M_SetStatus(stat.nState);	
	RETURN;
	
	
	///////////////////////////////////////////
	E_CRYO_BIN_CTRL_STATE.ACTIVE_SWITCHING_OFF:
	///////////////////////////////////////////
	//
	// Check for timeout
	timer(IN:=TRUE);
	IF timer.Q THEN
		// Stop the timer
		timer(IN:=FALSE);
		// Goto ERROR state
		stat.nState	:= E_CRYO_BIN_CTRL_STATE.ERROR;
	ELSIF	Actuator.stat.bError	THEN
		stat.nState	:= E_CRYO_BIN_CTRL_STATE.ERROR;
	ELSIF Actuator.stat.bOFF THEN
		// The actuator is OFF, transition completed.
		// Goto Active_Off.
		stat.nState	:= E_CRYO_BIN_CTRL_STATE.ACTIVE_OFF;
	END_IF
	M_SetStatus(stat.nState);	
	RETURN;
	
	/////////////////////////////////
	E_CRYO_BIN_CTRL_STATE.ERROR:
	/////////////////////////////////
	//
	M_User_TryRecovery();

END_CASE

METHOD M_Reset
VAR_INPUT
END_VAR
// By setting the bReset flag,
// The actuator will try to exit error state.
// In ERROR state, method M_User_TryRecovery() is executed.
bReset	:= TRUE;
END_METHOD

METHOD M_SetStatus
VAR_INPUT
	nState:	E_CRYO_BIN_CTRL_STATE;
END_VAR
stat.bActON		:= Actuator.stat.bON;
stat.bActOFF	:= Actuator.stat.bOFF;


CASE nState OF
	
	E_CRYO_BIN_CTRL_STATE.OFF:
	stat.bDone	:= TRUE;
	stat.bBusy	:= FALSE;
	stat.bError	:= FALSE;
	stat.bActive:= FALSE;
	stat.sState	:= 'OFF';
	
	E_CRYO_BIN_CTRL_STATE.ACTIVE_OFF:
	stat.bDone	:= TRUE;
	stat.bBusy	:= FALSE;
	stat.bError	:= FALSE;
	stat.bActive:= TRUE;
	stat.sState	:= 'ACTIVE_OFF';
	
	E_CRYO_BIN_CTRL_STATE.ACTIVE_ON:
	stat.bDone	:= TRUE;
	stat.bBusy	:= FALSE;
	stat.bError	:= FALSE;
	stat.bActive:= TRUE;
	stat.sState	:= 'ACTIVE_ON';
	
	E_CRYO_BIN_CTRL_STATE.ACTIVE_SWITCHING_ON:
	stat.bDone	:= FALSE;
	stat.bBusy	:= TRUE;
	stat.bError	:= FALSE;
	stat.bActive:= TRUE;
	stat.sState	:= 'ACTIVE_SWITCHING_ON...';
	
	E_CRYO_BIN_CTRL_STATE.ACTIVE_SWITCHING_OFF:
	stat.bDone	:= FALSE;
	stat.bBusy	:= TRUE;
	stat.bError	:= FALSE;
	stat.bActive:= TRUE;
	stat.sState	:= 'ACTIVE_SWITCHING_OFF...';
	
	E_CRYO_BIN_CTRL_STATE.ERROR:
	stat.bDone	:= TRUE;
	stat.bBusy	:= FALSE;
	stat.bError	:= TRUE;
	stat.bActive:= FALSE;
	stat.sState	:= 'ERROR';

END_CASE
END_METHOD

METHOD M_User_SetAction : INT
VAR_INPUT
END_VAR
// TODO USER
//
// This method implements the logic for controlling the actuator.
// The actuator can be a heater, valve, etc.
// There are two input values from sensors and two deltas for comparison.
//
// This example implements the heater control with the following assumptions:
//
// in_lrInput1 - Temperature of the Cryo Bench (B)
// in_lrInput2 - Temperature of the Detector (D). Coming from Lakeshore.
// in_lrPar1 - Delta [K] to turn the heater ON:  IF B < D - in_lrPar1
// in_lrPar2 - Delta [K] to turn the heater OFF: IF B > D - in_lrPar2
//
// in_lrDelta1 > in_lrDelta2, e.g. 10K > 4K.
//
IF	stat.nState = E_CRYO_BIN_CTRL_STATE.ACTIVE_OFF  OR  
	stat.nState = E_CRYO_BIN_CTRL_STATE.ACTIVE_ON THEN
(*	
	IF in_lrInput1 < in_lrInput2 - in_lrPar1 THEN
		// Activate the actuator
		M_User_SetOutput	:= E_CRYO_BIN_CTRL_ACTION.ON;
	ELSIF in_lrInput1 > in_lrInput2 - in_lrPar2 THEN
		// Dectivate the actuator
		M_User_SetOutput	:= E_CRYO_BIN_CTRL_ACTION.OFF;
	END_IF
*)
ELSE
	// Don't do anything
	M_User_SetAction	:= E_CRYO_BIN_CTRL_ACTION.NONE;
END_IF
END_METHOD

METHOD M_User_TryRecovery
VAR_INPUT
END_VAR
// TODO USER
// This is the default recovery routine.
// To be customided by the user, if needed.
//
IF bReset THEN
	// RESET the controller in order to try to clear error
	bReset	:= FALSE;	// Clear RESET flag
	
	// Start the timer
	timer(IN:=FALSE);
	timer(IN:=TRUE, PT:=T#5S);
	
	// Trigger action
	Actuator(in_bExecute:=FALSE);
	Actuator(in_bExecute:=TRUE, in_nCommand:=E_CRYO_BIN_ACT_CMD.OFF);
	
	// Goto SWITCHING_OFF state
	stat.nState	:= E_CRYO_BIN_CTRL_STATE.ACTIVE_SWITCHING_OFF;
	M_SetStatus(stat.nState);	
ELSIF NOT Actuator.stat.bError AND stat.bCtrlOK  THEN
	// Self recovery since everything seems to be OK now.
	// Goto NONE state.
	// From there proper state will be found and set.
	stat.nState	:= E_CRYO_BIN_CTRL_STATE.NONE;
	M_SetStatus(stat.nState);	
END_IF
END_METHOD

END_FUNCTION_BLOCK

// POUs/Actuators/FB_CRYO_CCC_CTRL
FUNCTION_BLOCK FB_CRYO_CCC_CTRL EXTENDS FB_CRYO_BIN_CTRL
VAR_INPUT
END_VAR
VAR_OUTPUT
END_VAR
VAR
	// Feedback from CCC
	{attribute 'OPC.UA.DA' := '0'}
	i_bOn				AT%I*:	BOOL;
	{attribute 'OPC.UA.DA' := '0'}
	i_bOverTemperature	AT%I*:	BOOL;
	{attribute 'OPC.UA.DA' := '0'}
	i_bUnderPressure	AT%I*:	BOOL;
END_VAR

// Set generic error if temperature inputs are not valid
IF i_bOn  AND  (i_bOverTemperature OR i_bUnderPressure) THEN
	stat.bCtrlOK	:= FALSE;
ELSE
	stat.bCtrlOK	:= TRUE;
END_IF

// Execute parent FB.
SUPER^();

METHOD M_User_SetAction : INT
VAR_INPUT
END_VAR
// TODO USER
//
// This method implements the logic for controlling a CCC.
//
// If the controller is Enabled, it should be ACTIVE_ON.
// If the controller is NOT Enabled, it should be OFF.
// 
//
IF	in_bEnable THEN
	M_User_SetAction	:= E_CRYO_BIN_CTRL_ACTION.ON;
ELSE
	M_User_SetAction	:= E_CRYO_BIN_CTRL_ACTION.OFF;
END_IF
END_METHOD

END_FUNCTION_BLOCK

// POUs/Actuators/FB_CRYO_CMD_OVERRIDE
FUNCTION_BLOCK FB_CRYO_CMD_OVERRIDE
VAR_INPUT
	in_bEnable:		BOOL;			// External ON/OFF command.
	in_bCorrEngCmd:	BOOL := FALSE;	// Correct active ENG command when switching to MANUAL Mode.
END_VAR
VAR_OUTPUT
	out_bEnable:	BOOL := FALSE;	// Resulting command
	out_bError:		BOOL := FALSE;	// Error flag (bug in SW implementation)
	out_bInterlock:	BOOL := FALSE;	// Flag if any command is prevented
	out_bWarning:	BOOL := FALSE;	// ENG command set to a not permitted command
	out_sMode:		STRING := '';	// Active Mode
	out_sStatus:	STRING := 'OK';	// Textual description in case of problems
END_VAR
VAR
	bAutoMode:		BOOL := TRUE;	// AUTO=true, MANUAL=false
	bEngMode:		BOOL := FALSE;	// Commissioning/Engineering mode. Ignores interlocks
	
	
	// Disable/enable manual control buttons
	bDisableBtnOn:	BOOL := FALSE;
	bDisableBtnOff:	BOOL := FALSE;

	// ON/OFF command permissions
	bPermitOn:		BOOL := TRUE;
	bPermitOff:		BOOL := TRUE;
	
	// Manual command
	bManualCmd:		BOOL := FALSE;
	
	// Reset interlocks (if possible)
	bReset:			BOOL := FALSE;
END_VAR

// Interlock is active if any command is not allowed
out_bInterlock	:= (NOT bPermitOn) OR (NOT bPermitOff);

// Both commands cannot be prevented at the same time ==> error
out_bError	:= (NOT bPermitOn) AND (NOT bPermitOff);

// This should never happen. Indicates error in the implementation.
IF out_bError	THEN
	out_sStatus	:= 'ERROR: Both commands prevented!';
	RETURN;
ELSE
	out_sStatus	:= 'OK';
END_IF


IF bAutoMode THEN
	out_sMode	:= 'AUTO';
	
	// There are no warnings in AUTO mode.
	out_bWarning:= FALSE;
	
	// Disable Manual control buttons
	bDisableBtnOn	:= TRUE;
	bDisableBtnOff	:= TRUE;
	
	// Only permitted commands can be set. Otherwise, error.
	IF in_bEnable AND NOT bPermitOn THEN
		// Impossible condition ==> error
		out_sStatus	:= 'ERROR: System command TRUE not permitted!';
		out_bError	:= TRUE;
		RETURN;
	ELSIF NOT in_bEnable AND NOT bPermitOff THEN
		// Impossible condition ==> error
		out_sStatus	:= 'ERROR: System command FALSE not permitted!';
		out_bError	:= TRUE;
		RETURN;
	END_IF
	
	// IN command =+> OUT command.
	bManualCmd	:= in_bEnable;
	out_bEnable	:= in_bEnable;

ELSIF bEngMode	THEN
	out_sMode	:= 'ENG';
	
	// No restrictions, no safety !!!
	// User responsible for damage caused by wrong/dangerous commands.

	// Enable both buttons.
	bDisableBtnOn	:= FALSE;
	bDisableBtnOff	:= FALSE;
	
	// Only set a warning if the user selects a command that the system doesn't allow.
	IF bManualCmd AND NOT bPermitOn THEN
		out_sStatus	:= 'WARNING: Command TRUE is not safe!';
		out_bWarning:= TRUE;
	ELSIF NOT bManualCmd AND NOT bPermitOff THEN
		out_sStatus	:= 'WARNING: Command FALSE is not safe!';
		out_bWarning:= TRUE;
	ELSE
		out_sStatus	:= 'OK';
		out_bWarning:= FALSE;
	END_IF

	// Assign user command to the output without any checks !!!
	out_bEnable		:= bManualCmd;

ELSE	// Manual mode.
	out_sMode	:= 'MANUAL';
	
	// Enable only permitted buttons.
	bDisableBtnOn	:= NOT bPermitOn;
	bDisableBtnOff	:= NOT bPermitOff;
	
	IF in_bCorrEngCmd	THEN
		// When exiting ENG Mode, if this flag is set, 
		// correct command set in ENG Mode if not permitted.
		IF	bManualCmd = TRUE   AND  NOT bPermitOn  THEN
			bManualCmd	:= FALSE;	// Set command to OFF
		ELSIF	bManualCmd = FALSE   AND  NOT bPermitOff  THEN
			bManualCmd	:= TRUE;	// Set command to ON
		END_IF
	END_IF

	// Only set a warning if the user selects a command that the system doesn't allow.
	IF bManualCmd AND NOT bPermitOn THEN
		out_sStatus	:= 'WARNING: Command TRUE is not safe!';
		out_bWarning:= TRUE;
	ELSIF NOT bManualCmd AND NOT bPermitOff THEN
		out_sStatus	:= 'WARNING: Command FALSE is not safe!';
		out_bWarning:= TRUE;
	ELSE
		out_sStatus	:= 'OK';
		out_bWarning:= FALSE;
	END_IF

	// Set the output command
	out_bEnable		:= bManualCmd;
END_IF

METHOD M_SetAllPermitted
VAR_INPUT
END_VAR
bPermitOn	:= TRUE;
bPermitOff	:= TRUE;
END_METHOD

METHOD M_SetPermissionOff
VAR_INPUT
	in_bPermit:	BOOL;
END_VAR
bPermitOff	:= in_bPermit;
END_METHOD

METHOD M_SetPermissionOn
VAR_INPUT
	in_bPermit:	BOOL;
END_VAR
bPermitOn	:= in_bPermit;
END_METHOD

METHOD M_SetPermissions
VAR_INPUT
	in_bPermitOn:	BOOL;
	in_bPermitOff:	BOOL;
END_VAR
bPermitOn	:= in_bPermitOn;
bPermitOff	:= in_bPermitOff;
END_METHOD

END_FUNCTION_BLOCK

// POUs/Actuators/FB_CRYO_GEN_CTRL_BASE
// Generic Controller
FUNCTION_BLOCK FB_CRYO_GEN_CTRL_BASE
VAR_INPUT
	in_bEnable:			BOOL := FALSE;	// Controller active while in_bEnable is TRUE
	in_nTimeout:		UDINT := 10000;	// Timeout for switching on/off [ms]. Default 10000.
	(*
		TODO USER: Add all specific input parameters, e.g.
		- Configuration parameters
		- External variables, e.g. temperature, pressure, etc.
	*)
END_VAR
VAR
	(*
		TODO USER: Add all system actuators, variables and I/O signals, e.g.
		
		{attribute 'OPC.UA.DA' := '1'}
		Actuator:	FB_CRYO_BIN_ACT;	// Heater, valve, etc.
	*)
	
	{attribute 'OPC.UA.DA' := '0'}
	statRef:	REFERENCE TO T_CRYO_GEN_CTRL_STATUS_BASE;

	(*
		TODO USER:	Add a 'stat' structure.
					It can be the T_CRYO_GEN_CTRL_STATUS or a struct that EXTENDS T_CRYO_GEN_CTRL_STATUS.
					For example:
						stat:	T_CRYO_BIN_CTRL_STATUS;
	*)
	
	nEvent:		E_CRYO_GEN_CTRL_EVENT := E_CRYO_GEN_CTRL_EVENT.NONE;

	{attribute 'OPC.UA.DA' := '0'}
	timer:		TON;		// Timer for commands
	
	{attribute 'OPC.UA.DA' := '0'}
	trgEnable:	R_TRIG;		// Rising trigger of in_bEnable
	
	// This flag will be set once M_Configure() is executed.
	bConfigured:	BOOL := FALSE;
END_VAR

// Don't do anything until the controller is configured
IF NOT bConfigured THEN
	M_Configure();
	RETURN;
END_IF

// Increment cycle counter
statRef.nCycleCounter := statRef.nCycleCounter + 1;



M_ReadInputs();


M_ExecuteActuators();


M_SetStatus();


M_CheckForEvents();


M_ProcessEvents();

METHOD M_ActionOffExecute
VAR_INPUT
END_VAR
//
// In this method the user shall turn off the actuator(s) such as valves, heaters, coolers, etc.
// Normally this is done by setting the in_bEnable flag of the actuator to FALSE.
// In the corresponding Activity M_ActivitySwitchingOff(), the completion of the OFF command shall be checked.
//
timer(IN:=FALSE);	// Reset Timer - mandatory!
END_METHOD

METHOD M_ActionOnExecute
VAR_INPUT
END_VAR
// In this method the user shall turn on the actuator(s) such as valves, heaters, coolers, etc.
// Normally this is done by setting the in_bEnable flag of the actuator to TRUE.
// In the corresponding Activity M_ActivitySwitchingOn(), the completion of the ON command shall be checked.
timer(IN:=FALSE);	// Reset Timer
END_METHOD

METHOD M_ActivitySwitchingOff : BOOL
VAR_INPUT
END_VAR
// In this method the user shall wait until the actuator is turned OFF.
// The actuator state is available in the status structure.
// When complete, the method shall return TRUE, otherwise FALSE.


// Dummy implementation.
// Complete after 5 sec.
//
timer(IN:=TRUE, PT:=UDINT_TO_TIME(in_nTimeout));
	
IF timer.ET >= T#5S THEN
	M_ActivitySwitchingOff := TRUE;
ELSE
	M_ActivitySwitchingOff := FALSE;
END_IF
END_METHOD

METHOD M_ActivitySwitchingOn : BOOL
VAR_INPUT
END_VAR
// In this method the user shall wait until the actuator is turned ON.
// The actuator state is available in the status structure.
// When complete, the method shall return TRUE, otherwise FALSE.


// Dummy implementation.
// Complete after 5 sec.
//
timer(IN:=TRUE, PT:=UDINT_TO_TIME(in_nTimeout));
	
IF timer.ET >= T#5S THEN
	M_ActivitySwitchingOn := TRUE;
ELSE
	M_ActivitySwitchingOn := FALSE;
END_IF
END_METHOD

METHOD M_CheckForEvents
VAR_INPUT
END_VAR
VAR
	nEventTmp:	E_CRYO_GEN_CTRL_EVENT := E_CRYO_GEN_CTRL_EVENT.NONE;
END_VAR
// TODO USER
//

nEventTmp	:= E_CRYO_GEN_CTRL_EVENT.NONE;

// Check for the Enable trigger
trgEnable(CLK := in_bEnable);


CASE statRef.nState OF
	/////////////////////////////////
	E_CRYO_BIN_CTRL_STATE.NONE:
	/////////////////////////////////
	//
	// This is the state on power-up.
	statRef.nState	:= E_CRYO_BIN_CTRL_STATE.OFF;
	

	/////////////////////////////////
	E_CRYO_BIN_CTRL_STATE.OFF:
	/////////////////////////////////
	//
	IF	trgEnable.Q  THEN
		nEventTmp	:= E_CRYO_GEN_CTRL_EVENT.ENABLE;
	END_IF
	
	
	/////////////////////////////////
	E_CRYO_BIN_CTRL_STATE.ACTIVE_OFF:
	/////////////////////////////////
	//
	IF NOT in_bEnable  THEN
		// Goto Off.
		//
		nEventTmp	:= E_CRYO_GEN_CTRL_EVENT.DISABLE;
	ELSIF M_ControlLoop() = TRUE THEN
		nEventTmp	:= E_CRYO_GEN_CTRL_EVENT.ON;
	END_IF
	
	
	//////////////////////////////////////////
	E_CRYO_BIN_CTRL_STATE.ACTIVE_SWITCHING_ON:
	//////////////////////////////////////////
	//
	IF NOT in_bEnable  THEN
		// Goto ACTIVE_OF first.
		//
		nEventTmp	:= E_CRYO_GEN_CTRL_EVENT.OFF;
	ELSIF timer.Q THEN
		nEventTmp	:= E_CRYO_GEN_CTRL_EVENT.ERROR;
	ELSIF M_ControlLoop() = FALSE THEN
		nEventTmp	:= E_CRYO_GEN_CTRL_EVENT.OFF;
	ELSIF M_ActivitySwitchingOn() THEN
		nEventTmp	:= E_CRYO_GEN_CTRL_EVENT.IS_ON;
	END_IF
	

	//////////////////////////////////////////
	E_CRYO_BIN_CTRL_STATE.ACTIVE_ON:
	//////////////////////////////////////////
	//
	IF NOT in_bEnable  THEN
		// Goto ACTIVE_OFF first.
		//
		nEventTmp	:= E_CRYO_GEN_CTRL_EVENT.OFF;
	ELSIF M_ControlLoop() = FALSE THEN
		nEventTmp	:= E_CRYO_GEN_CTRL_EVENT.OFF;
	END_IF
	

	///////////////////////////////////////////
	E_CRYO_BIN_CTRL_STATE.ACTIVE_SWITCHING_OFF:
	///////////////////////////////////////////
	//
	IF NOT in_bEnable  THEN
		// Goto Off.
		//
		nEventTmp	:= E_CRYO_GEN_CTRL_EVENT.DISABLE;
	ELSIF timer.Q THEN
		nEventTmp	:= E_CRYO_GEN_CTRL_EVENT.ERROR;
	ELSIF M_ControlLoop() = TRUE THEN
		nEventTmp	:= E_CRYO_GEN_CTRL_EVENT.ON;
	ELSIF M_ActivitySwitchingOff() THEN
		nEventTmp	:= E_CRYO_GEN_CTRL_EVENT.IS_OFF;
	END_IF
	

	/////////////////////////////////
	E_CRYO_BIN_CTRL_STATE.ERROR:
	/////////////////////////////////
	//
	IF	trgEnable.Q  THEN
		nEventTmp	:= E_CRYO_GEN_CTRL_EVENT.ENABLE;
	END_IF
	
END_CASE

nEvent	:= nEventTmp;
END_METHOD

METHOD M_Configure
VAR_INPUT
END_VAR
// Configure the system and set the bConfigured flag to TRUE.

(*
	TODO USER: 
	- Set references to extended structures. e.g.
	- Configure the system, if any.
	
	MUST be the very first line!!!
	     statRef REF=stat;
*)

// The system has been configured
bConfigured := TRUE;
END_METHOD

METHOD M_ControlLoop : BOOL
VAR_INPUT
END_VAR
VAR_INST
	timerDummy:	TON;	// Dummy timer
	nDummy:		UDINT;	// Dummy counter
END_VAR
// Dummy implementation of the control loop.
// The return value says if the loop should be ACTIVE/TRUE or INACTIVE/FALSE

IF nDummy = 0 THEN
	timerDummy(IN:=FALSE);	// Reset timer
END_IF
nDummy	:= nDummy + 1;

timerDummy(IN:=TRUE, PT:=T#10S);

CASE statRef.nState OF
	E_CRYO_BIN_CTRL_STATE.ACTIVE_SWITCHING_OFF,
	E_CRYO_BIN_CTRL_STATE.ACTIVE_OFF:
		IF timerDummy.Q THEN
			nDummy := 0;
			// This will create ON event.
			M_ControlLoop	:= TRUE;
		ELSE
			// Remain OFF
			M_ControlLoop	:= FALSE;
		END_IF
	E_CRYO_BIN_CTRL_STATE.ACTIVE_SWITCHING_ON,
	E_CRYO_BIN_CTRL_STATE.ACTIVE_ON:
		IF timerDummy.Q THEN
			nDummy := 0;
			// This will create OFF event.
			M_ControlLoop	:= FALSE;
		ELSE
			// Remain ON
			M_ControlLoop	:= TRUE;
		END_IF
	ELSE
		M_ControlLoop	:= FALSE;
END_CASE
END_METHOD

METHOD M_ExecuteActuators
VAR_INPUT
END_VAR
(*
	TODO USER: Execute all actuators, e.g. valve, heater, etc.


// Example: Execute Actuator FB instance
Actuator(
	in_nFeedback		:= in_nFeedback,
	in_nTimeout			:= in_nTimeout,
	in_bActiveLowCtrl	:= in_bActiveLowCtrl,
	in_bActiveLowStat	:= in_bActiveLowStat);


*)
END_METHOD

METHOD M_IsError : BOOL
VAR_INPUT
END_VAR
(*
	TODO USER: Do all the checks and return TRUE if error.
	Otherwise, return FALSE (no error).
*)

M_IsError	:= FALSE;
END_METHOD

METHOD M_ProcessEvents
VAR_INPUT
END_VAR
// TODO USER
//


CASE statRef.nState OF
	/////////////////////////////////
	E_CRYO_BIN_CTRL_STATE.NONE:
	/////////////////////////////////
	//
	// Nothing to do.
	;
	

	/////////////////////////////////
	E_CRYO_BIN_CTRL_STATE.OFF:
	/////////////////////////////////
	//
	IF	nEvent = E_CRYO_GEN_CTRL_EVENT.ENABLE  THEN
		// Activate the control loop.
		// Goto Active_Off first.
		//
		M_ActionOffExecute();		
		// Set next state
		statRef.nState	:= E_CRYO_BIN_CTRL_STATE.ACTIVE_SWITCHING_OFF;
	END_IF
	
	
	/////////////////////////////////
	E_CRYO_BIN_CTRL_STATE.ACTIVE_OFF:
	/////////////////////////////////
	//
	IF	nEvent = E_CRYO_GEN_CTRL_EVENT.DISABLE  THEN
		// Goto Off.
		//
		// Set next state
		statRef.nState	:= E_CRYO_BIN_CTRL_STATE.OFF;
	ELSIF nEvent = E_CRYO_GEN_CTRL_EVENT.ON THEN
		M_ActionOnExecute();
		// Set next state
		statRef.nState	:= E_CRYO_BIN_CTRL_STATE.ACTIVE_SWITCHING_ON;
	END_IF
	
	
	//////////////////////////////////////////
	E_CRYO_BIN_CTRL_STATE.ACTIVE_SWITCHING_ON:
	//////////////////////////////////////////
	//
	// Check for timeout
	IF timer.Q THEN
		// Goto ERROR state
		statRef.nState	:= E_CRYO_BIN_CTRL_STATE.ERROR;
	ELSIF nEvent = E_CRYO_GEN_CTRL_EVENT.OFF THEN
		M_ActionOffExecute();
		// Set next state
		statRef.nState	:= E_CRYO_BIN_CTRL_STATE.ACTIVE_SWITCHING_OFF;
	ELSIF M_ActivitySwitchingOn() THEN
		statRef.nState	:= E_CRYO_BIN_CTRL_STATE.ACTIVE_ON;
	END_IF
	

	/////////////////////////////////
	E_CRYO_BIN_CTRL_STATE.ACTIVE_ON:
	/////////////////////////////////
	//
	IF	nEvent = E_CRYO_GEN_CTRL_EVENT.DISABLE  THEN
		// Goto Off.
		//
		M_ActionOffExecute();
		// Set next state
		statRef.nState	:= E_CRYO_BIN_CTRL_STATE.ACTIVE_SWITCHING_OFF;
	ELSIF nEvent = E_CRYO_GEN_CTRL_EVENT.OFF THEN
		M_ActionOffExecute();
		// Set next state
		statRef.nState	:= E_CRYO_BIN_CTRL_STATE.ACTIVE_SWITCHING_OFF;
	END_IF
	
	
	///////////////////////////////////////////
	E_CRYO_BIN_CTRL_STATE.ACTIVE_SWITCHING_OFF:
	///////////////////////////////////////////
	//
	// Check for timeout
	IF timer.Q THEN
		// Goto ERROR state
		statRef.nState	:= E_CRYO_BIN_CTRL_STATE.ERROR;
	ELSIF nEvent = E_CRYO_GEN_CTRL_EVENT.ON THEN
		M_ActionOnExecute();
		// Set next state
		statRef.nState	:= E_CRYO_BIN_CTRL_STATE.ACTIVE_SWITCHING_ON;
	ELSIF M_ActivitySwitchingOff() THEN
		statRef.nState	:= E_CRYO_BIN_CTRL_STATE.ACTIVE_OFF;
	END_IF

	
	/////////////////////////////////
	E_CRYO_BIN_CTRL_STATE.ERROR:
	/////////////////////////////////
	//
	IF	nEvent = E_CRYO_GEN_CTRL_EVENT.ENABLE  THEN
		// Activate the control loop.
		// Goto Active_Off first.
		//
		// Set next state
		statRef.nState	:= E_CRYO_BIN_CTRL_STATE.ACTIVE_OFF;
	END_IF
	
END_CASE


// If error, goto ERROR state.
IF M_IsError() THEN
	statRef.nState	:= E_CRYO_BIN_CTRL_STATE.ERROR;
END_IF

// Set status
M_SetStatus();
END_METHOD

METHOD M_ReadInputs
VAR_INPUT
END_VAR
(*
	TODO USER: Read all inputs and assign values to variables.
	Inputs can be pressure, temperature, etc.
*)
END_METHOD

METHOD M_SetStatus
VAR_INPUT
END_VAR
CASE statRef.nState OF
	
	E_CRYO_BIN_CTRL_STATE.OFF:
	statRef.bDone	:= TRUE;
	statRef.bBusy	:= FALSE;
	statRef.bError	:= FALSE;
	statRef.bActive	:= FALSE;
	statRef.sState	:= 'OFF';
	
	E_CRYO_BIN_CTRL_STATE.ACTIVE_OFF:
	statRef.bDone	:= TRUE;
	statRef.bBusy	:= FALSE;
	statRef.bError	:= FALSE;
	statRef.bActive	:= TRUE;
	statRef.sState	:= 'ACTIVE_OFF';
	
	E_CRYO_BIN_CTRL_STATE.ACTIVE_ON:
	statRef.bDone	:= TRUE;
	statRef.bBusy	:= FALSE;
	statRef.bError	:= FALSE;
	statRef.bActive	:= TRUE;
	statRef.sState	:= 'ACTIVE_ON';
	
	E_CRYO_BIN_CTRL_STATE.ACTIVE_SWITCHING_ON:
	statRef.bDone	:= FALSE;
	statRef.bBusy	:= TRUE;
	statRef.bError	:= FALSE;
	statRef.bActive	:= TRUE;
	statRef.sState	:= 'ACTIVE_SWITCHING_ON...';
	
	E_CRYO_BIN_CTRL_STATE.ACTIVE_SWITCHING_OFF:
	statRef.bDone	:= FALSE;
	statRef.bBusy	:= TRUE;
	statRef.bError	:= FALSE;
	statRef.bActive	:= TRUE;
	statRef.sState	:= 'ACTIVE_SWITCHING_OFF...';
	
	E_CRYO_BIN_CTRL_STATE.ERROR:
	statRef.bDone	:= TRUE;
	statRef.bBusy	:= FALSE;
	statRef.bError	:= TRUE;
	statRef.bActive	:= FALSE;
	statRef.sState	:= 'ERROR';

END_CASE

IF NOT statRef.bError THEN
	statRef.sError := 'OK';
END_IF
END_METHOD

END_FUNCTION_BLOCK

// POUs/Actuators/FB_CRYO_HEATER_CTRL
FUNCTION_BLOCK FB_CRYO_HEATER_CTRL EXTENDS FB_CRYO_BIN_CTRL
VAR_INPUT
	// Two input values for comparison
	in_lrTemp1:		LREAL;	// Lowest temperature in  cryostat
	in_lrTemp2:		LREAL;	// Detector temperature.
	// Input values Valid flag
	in_bValidTemp1:	BOOL;
	in_bValidTemp2:	BOOL;
	// Two parameters for decision making
	// Delat-T SetPoint between Detector and Coldbench during WarmUp
	in_lrDelta_Low:		LREAL	:= 10.0;
	// Delat-T SetPoint between Detector and Coldbench during WarmUp	
	in_lrDelta_High:	LREAL	:= 5.0;

END_VAR
VAR_OUTPUT
END_VAR
VAR
END_VAR

// Set generic error if temperature inputs are not valid
IF NOT in_bValidTemp1 OR NOT in_bValidTemp2  THEN
	stat.bCtrlOK	:= FALSE;
ELSE
	stat.bCtrlOK	:= TRUE;
END_IF

// Execute parent FB.
SUPER^();

